LIN {X 0,Y 401.052,Z 702.53,A -85,B 0,C 180,E1 10289.297,E2 10289.297} C_VEL
LIN {X 0,Y 401.045,Z 702.53,A -85,B 0,C 180,E1 10294.373,E2 10294.373} C_VEL
LIN {X 0,Y 400.94,Z 702.53,A -85,B 0,C 180,E1 10301.171,E2 10301.171} C_VEL
LIN {X 0,Y 400.996,Z 702.775,A -85,B 0,C 180,E1 10303.002,E2 10303.002} C_VEL
LIN {X 0,Y 403.697,Z 708.428,A -85,B 0,C 180,E1 10303.533,E2 10303.533} C_VEL
LIN {X 0,Y 424.245,Z 745.989,A -85,B 0,C 180,E1 10307.047,E2 10307.047} C_VEL
LIN {X 0,Y 435.386,Z 772.98,A -85,B 0,C 180,E1 10309.087,E2 10309.087} C_VEL
LIN {X 0,Y 431.382,Z 812.336,A -85,B 0,C 180,E1 10310.627,E2 10310.627} C_VEL
LIN {X 0,Y 426.154,Z 850.577,A -85,B 0,C 180,E1 10312.988,E2 10312.988} C_VEL
LIN {X 0,Y 420.465,Z 885.103,A -85,B 0,C 180,E1 10316.006,E2 10316.006} C_VEL
LIN {X 0,Y 414.847,Z 916.19,A -85,B 0,C 180,E1 10319.673,E2 10319.673} C_VEL
LIN {X 0,Y 409.958,Z 944.249,A -85,B 0,C 180,E1 10324.079,E2 10324.079} C_VEL
LIN {X 0,Y 406.182,Z 967.928,A -85,B 0,C 180,E1 10329.048,E2 10329.048} C_VEL
LIN {X 0,Y 405.097,Z 975.872,A -85,B 0,C 180,E1 10331.112,E2 10331.112} C_VEL
LIN {X 0,Y 400.257,Z 983.264,A -85,B 0,C 180,E1 10333.268,E2 10333.268} C_VEL
LIN {X 0,Y 395.701,Z 989.61,A -85,B 0,C 180,E1 10335.54,E2 10335.54} C_VEL
LIN {X 0,Y 395,Z 999.376,A -85,B 0,C 180,E1 10340.101,E2 10340.101} C_VEL
LIN {X 0,Y 394.611,Z 1006.165,A -85,B 0,C 180,E1 10345.613,E2 10345.613} C_VEL
LIN {X 0,Y 394.714,Z 1007.908,A -85,B 0,C 180,E1 10350,E2 10350} C_VEL
LIN {X 0,Y 394.611,Z 1006.224,A -85,B 0,C 180,E1 10354.386,E2 10354.386} C_VEL
LIN {X 0,Y 394.945,Z 999.516,A -85,B 0,C 180,E1 10359.9,E2 10359.9} C_VEL
LIN {X 0,Y 395.941,Z 987.247,A -85,B 0,C 180,E1 10365.473,E2 10365.473} C_VEL
LIN {X 0,Y 398.331,Z 968.706,A -85,B 0,C 180,E1 10371.093,E2 10371.093} C_VEL
LIN {X 0,Y 402.279,Z 945.825,A -85,B 0,C 180,E1 10376.109,E2 10376.109} C_VEL
LIN {X 0,Y 407.443,Z 918.337,A -85,B 0,C 180,E1 10380.614,E2 10380.614} C_VEL
LIN {X 0,Y 413.535,Z 886.366,A -85,B 0,C 180,E1 10384.518,E2 10384.518} C_VEL
LIN {X 0,Y 419.816,Z 850.978,A -85,B 0,C 180,E1 10387.666,E2 10387.666} C_VEL
LIN {X 0,Y 425.063,Z 815.15,A -85,B 0,C 180,E1 10389.921,E2 10389.921} C_VEL
LIN {X 0,Y 429.128,Z 778.016,A -85,B 0,C 180,E1 10391.452,E2 10391.452} C_VEL
LIN {X 0,Y 428.274,Z 771.788,A -85,B 0,C 180,E1 10391.794,E2 10391.794} C_VEL
LIN {X 0,Y 411.741,Z 736.797,A -85,B 0,C 180,E1 10394.654,E2 10394.654} C_VEL
LIN {X 0,Y 393.146,Z 703.935,A -85,B 0,C 180,E1 10397.845,E2 10397.845} C_VEL
LIN {X 0,Y 392.991,Z 702.53,A -85,B 0,C 180,E1 10398.003,E2 10398.003} C_VEL
LIN {X 0,Y 393.035,Z 702.53,A -85,B 0,C 180,E1 10404.824,E2 10404.824} C_VEL
LIN {X 0,Y 393.229,Z 702.53,A -85,B 0,C 180,E1 10410.062,E2 10410.062} C_VEL
LIN {X 0,Y 393.395,Z 702.53,A -85,B 0,C 180,E1 10417.43,E2 10417.43} C_VEL
LIN {X 0,Y 393.756,Z 702.53,A -85,B 0,C 180,E1 10424.424,E2 10424.424} C_VEL
LIN {X 0,Y 394.01,Z 702.53,A -85,B 0,C 180,E1 10431.172,E2 10431.172} C_VEL
LIN {X 0,Y 394.34,Z 702.53,A -85,B 0,C 180,E1 10437.79,E2 10437.79} C_VEL
LIN {X 0,Y 394.238,Z 702.53,A -85,B 0,C 180,E1 10444.372,E2 10444.372} C_VEL
LIN {X 0,Y 393.912,Z 702.53,A -85,B 0,C 180,E1 10451.022,E2 10451.022} C_VEL
LIN {X 0,Y 393.605,Z 702.53,A -85,B 0,C 180,E1 10457.838,E2 10457.838} C_VEL
LIN {X 0,Y 393.332,Z 702.53,A -85,B 0,C 180,E1 10464.936,E2 10464.936} C_VEL
LIN {X 0,Y 393.129,Z 702.53,A -85,B 0,C 180,E1 10472.477,E2 10472.477} C_VEL
LIN {X 0,Y 393.096,Z 702.53,A -85,B 0,C 180,E1 10479.847,E2 10479.847} C_VEL
LIN {X 0,Y 392.99,Z 702.53,A -85,B 0,C 180,E1 10486.81,E2 10486.81} C_VEL
LIN {X 0,Y 393.02,Z 702.53,A -85,B 0,C 180,E1 10493.688,E2 10493.688} C_VEL
LIN {X 0,Y 393.251,Z 702.53,A -85,B 0,C 180,E1 10500.076,E2 10500.076} C_VEL
LIN {X 0,Y 393.474,Z 702.53,A -85,B 0,C 180,E1 10507.449,E2 10507.449} C_VEL
LIN {X 0,Y 393.781,Z 702.53,A -85,B 0,C 180,E1 10515.001,E2 10515.001} C_VEL
LIN {X 0,Y 393.859,Z 703.393,A -85,B 0,C 180,E1 10515.424,E2 10515.424} C_VEL
LIN {X 0,Y 412.86,Z 740.827,A -85,B 0,C 180,E1 10519.002,E2 10519.002} C_VEL
LIN {X 0,Y 422.422,Z 766.343,A -85,B 0,C 180,E1 10521.39,E2 10521.39} C_VEL
LIN {X 0,Y 417.672,Z 802.69,A -85,B 0,C 180,E1 10523.68,E2 10523.68} C_VEL
LIN {X 0,Y 412.384,Z 834.554,A -85,B 0,C 180,E1 10526.591,E2 10526.591} C_VEL
LIN {X 0,Y 406.978,Z 863.399,A -85,B 0,C 180,E1 10530.239,E2 10530.239} C_VEL
LIN {X 0,Y 401.875,Z 889.304,A -85,B 0,C 180,E1 10534.775,E2 10534.775} C_VEL
LIN {X 0,Y 398.263,Z 909.402,A -85,B 0,C 180,E1 10539.735,E2 10539.735} C_VEL
LIN {X 0,Y 396.131,Z 923.775,A -85,B 0,C 180,E1 10544.89,E2 10544.89} C_VEL
LIN {X 0,Y 395.152,Z 932.764,A -85,B 0,C 180,E1 10550.103,E2 10550.103} C_VEL
LIN {X 0,Y 394.324,Z 936.627,A -85,B 0,C 180,E1 10554.895,E2 10554.895} C_VEL
LIN {X 0,Y 394.397,Z 936.365,A -85,B 0,C 180,E1 10559.829,E2 10559.829} C_VEL
LIN {X 0,Y 395.362,Z 931.57,A -85,B 0,C 180,E1 10564.927,E2 10564.927} C_VEL
LIN {X 0,Y 396.711,Z 920.884,A -85,B 0,C 180,E1 10570.511,E2 10570.511} C_VEL
LIN {X 0,Y 399.154,Z 906.168,A -85,B 0,C 180,E1 10575.371,E2 10575.371} C_VEL
LIN {X 0,Y 403.025,Z 886.025,A -85,B 0,C 180,E1 10580.064,E2 10580.064} C_VEL
LIN {X 0,Y 408.334,Z 860.251,A -85,B 0,C 180,E1 10584.393,E2 10584.393} C_VEL
LIN {X 0,Y 414.18,Z 830.081,A -85,B 0,C 180,E1 10588.051,E2 10588.051} C_VEL
LIN {X 0,Y 419.598,Z 797.291,A -85,B 0,C 180,E1 10590.879,E2 10590.879} C_VEL
LIN {X 0,Y 423.349,Z 767.496,A -85,B 0,C 180,E1 10592.719,E2 10592.719} C_VEL
LIN {X 0,Y 410.879,Z 735.408,A -85,B 0,C 180,E1 10595.919,E2 10595.919} C_VEL
LIN {X 0,Y 394.941,Z 706.911,A -85,B 0,C 180,E1 10599.107,E2 10599.107} C_VEL
LIN {X 0,Y 393.602,Z 702.53,A -85,B 0,C 180,E1 10599.553,E2 10599.553} C_VEL
LIN {X 0,Y 393.925,Z 702.53,A -85,B 0,C 180,E1 10606.733,E2 10606.733} C_VEL
LIN {X 0,Y 394.164,Z 702.53,A -85,B 0,C 180,E1 10613.424,E2 10613.424} C_VEL
LIN {X 0,Y 394.433,Z 702.53,A -85,B 0,C 180,E1 10620.018,E2 10620.018} C_VEL
LIN {X 0,Y 394.167,Z 702.53,A -85,B 0,C 180,E1 10626.611,E2 10626.611} C_VEL
LIN {X 0,Y 393.791,Z 702.53,A -85,B 0,C 180,E1 10633.307,E2 10633.307} C_VEL
LIN {X 0,Y 393.496,Z 702.53,A -85,B 0,C 180,E1 10640.204,E2 10640.204} C_VEL
LIN {X 0,Y 393.162,Z 702.53,A -85,B 0,C 180,E1 10647.437,E2 10647.437} C_VEL
LIN {X 0,Y 393.102,Z 702.53,A -85,B 0,C 180,E1 10652.521,E2 10652.521} C_VEL
LIN {X 0,Y 393.103,Z 702.53,A -85,B 0,C 180,E1 10659.847,E2 10659.847} C_VEL
LIN {X 0,Y 393.027,Z 702.53,A -85,B 0,C 180,E1 10661.782,E2 10661.782} C_VEL
LIN {X 0,Y 395.507,Z 708.258,A -85,B 0,C 180,E1 10662.321,E2 10662.321} C_VEL
LIN {X 0,Y 413.841,Z 740.209,A -85,B 0,C 180,E1 10665.645,E2 10665.645} C_VEL
LIN {X 0,Y 428.982,Z 774.179,A -85,B 0,C 180,E1 10668.462,E2 10668.462} C_VEL
LIN {X 0,Y 424.791,Z 813.732,A -85,B 0,C 180,E1 10670.072,E2 10670.072} C_VEL
LIN {X 0,Y 419.489,Z 850.623,A -85,B 0,C 180,E1 10672.403,E2 10672.403} C_VEL
LIN {X 0,Y 413.587,Z 884.412,A -85,B 0,C 180,E1 10675.4,E2 10675.4} C_VEL
LIN {X 0,Y 407.742,Z 915.374,A -85,B 0,C 180,E1 10679.102,E2 10679.102} C_VEL
LIN {X 0,Y 402.477,Z 943.473,A -85,B 0,C 180,E1 10683.582,E2 10683.582} C_VEL
LIN {X 0,Y 398.489,Z 967.095,A -85,B 0,C 180,E1 10688.624,E2 10688.624} C_VEL
LIN {X 0,Y 396.091,Z 985.35,A -85,B 0,C 180,E1 10693.966,E2 10693.966} C_VEL
LIN {X 0,Y 395.701,Z 989.61,A -85,B 0,C 180,E1 10695.54,E2 10695.54} C_VEL
LIN {X 0,Y 394.194,Z 992.52,A -85,B 0,C 180,E1 10696.72,E2 10696.72} C_VEL
LIN {X 0,Y 387.214,Z 998.831,A -85,B 0,C 180,E1 10700.006,E2 10700.006} C_VEL
LIN {X 0,Y 387.072,Z 999.295,A -85,B 0,C 180,E1 10700.323,E2 10700.323} C_VEL
LIN {X 0,Y 386.742,Z 1005.449,A -85,B 0,C 180,E1 10705.524,E2 10705.524} C_VEL
LIN {X 0,Y 386.851,Z 1007.204,A -85,B 0,C 180,E1 10710,E2 10710} C_VEL
LIN {X 0,Y 386.743,Z 1005.522,A -85,B 0,C 180,E1 10714.475,E2 10714.475} C_VEL
LIN {X 0,Y 387.089,Z 998.806,A -85,B 0,C 180,E1 10720.103,E2 10720.103} C_VEL
LIN {X 0,Y 388.126,Z 986.517,A -85,B 0,C 180,E1 10725.792,E2 10725.792} C_VEL
LIN {X 0,Y 390.553,Z 968.854,A -85,B 0,C 180,E1 10731.294,E2 10731.294} C_VEL
LIN {X 0,Y 394.713,Z 946.035,A -85,B 0,C 180,E1 10736.443,E2 10736.443} C_VEL
LIN {X 0,Y 399.964,Z 919.435,A -85,B 0,C 180,E1 10740.934,E2 10740.934} C_VEL
LIN {X 0,Y 406.318,Z 887.704,A -85,B 0,C 180,E1 10744.929,E2 10744.929} C_VEL
LIN {X 0,Y 412.869,Z 852.832,A -85,B 0,C 180,E1 10748.128,E2 10748.128} C_VEL
LIN {X 0,Y 418.434,Z 816.703,A -85,B 0,C 180,E1 10750.477,E2 10750.477} C_VEL
LIN {X 0,Y 422.744,Z 779.639,A -85,B 0,C 180,E1 10752.058,E2 10752.058} C_VEL
LIN {X 0,Y 421.436,Z 773.287,A -85,B 0,C 180,E1 10752.464,E2 10752.464} C_VEL
LIN {X 0,Y 405.117,Z 738.587,A -85,B 0,C 180,E1 10755.43,E2 10755.43} C_VEL
LIN {X 0,Y 385.128,Z 703.353,A -85,B 0,C 180,E1 10759.006,E2 10759.006} C_VEL
LIN {X 0,Y 385.086,Z 702.53,A -85,B 0,C 180,E1 10759.18,E2 10759.18} C_VEL
LIN {X 0,Y 385.15,Z 702.53,A -85,B 0,C 180,E1 10766.722,E2 10766.722} C_VEL
LIN {X 0,Y 385.311,Z 702.53,A -85,B 0,C 180,E1 10771.955,E2 10771.955} C_VEL
LIN {X 0,Y 385.568,Z 702.53,A -85,B 0,C 180,E1 10779.362,E2 10779.362} C_VEL
LIN {X 0,Y 385.931,Z 702.53,A -85,B 0,C 180,E1 10786.416,E2 10786.416} C_VEL
LIN {X 0,Y 386.238,Z 702.53,A -85,B 0,C 180,E1 10793.252,E2 10793.252} C_VEL
LIN {X 0,Y 386.529,Z 702.53,A -85,B 0,C 180,E1 10799.982,E2 10799.982} C_VEL
LIN {X 0,Y 386.294,Z 702.53,A -85,B 0,C 180,E1 10806.71,E2 10806.71} C_VEL
LIN {X 0,Y 385.902,Z 702.53,A -85,B 0,C 180,E1 10813.548,E2 10813.548} C_VEL
LIN {X 0,Y 385.558,Z 702.53,A -85,B 0,C 180,E1 10820.601,E2 10820.601} C_VEL
LIN {X 0,Y 385.293,Z 702.53,A -85,B 0,C 180,E1 10828.006,E2 10828.006} C_VEL
LIN {X 0,Y 385.138,Z 702.53,A -85,B 0,C 180,E1 10835.963,E2 10835.963} C_VEL
LIN {X 0,Y 385.054,Z 702.53,A -85,B 0,C 180,E1 10841.875,E2 10841.875} C_VEL
LIN {X 0,Y 384.996,Z 702.53,A -85,B 0,C 180,E1 10848.216,E2 10848.216} C_VEL
LIN {X 0,Y 385.102,Z 702.53,A -85,B 0,C 180,E1 10855.323,E2 10855.323} C_VEL
LIN {X 0,Y 385.351,Z 702.53,A -85,B 0,C 180,E1 10861.971,E2 10861.971} C_VEL
LIN {X 0,Y 385.614,Z 702.53,A -85,B 0,C 180,E1 10869.379,E2 10869.379} C_VEL
LIN {X 0,Y 385.816,Z 702.53,A -85,B 0,C 180,E1 10874.301,E2 10874.301} C_VEL
LIN {X 0,Y 388.288,Z 708.228,A -85,B 0,C 180,E1 10874.797,E2 10874.797} C_VEL
LIN {X 0,Y 405.008,Z 740.357,A -85,B 0,C 180,E1 10878.064,E2 10878.064} C_VEL
LIN {X 0,Y 415.924,Z 768.941,A -85,B 0,C 180,E1 10880.868,E2 10880.868} C_VEL
LIN {X 0,Y 410.983,Z 804.002,A -85,B 0,C 180,E1 10883.128,E2 10883.128} C_VEL
LIN {X 0,Y 405.406,Z 836.162,A -85,B 0,C 180,E1 10886.132,E2 10886.132} C_VEL
LIN {X 0,Y 399.504,Z 865.889,A -85,B 0,C 180,E1 10890,E2 10890} C_VEL
LIN {X 0,Y 394.476,Z 890.181,A -85,B 0,C 180,E1 10894.388,E2 10894.388} C_VEL
LIN {X 0,Y 390.81,Z 909.432,A -85,B 0,C 180,E1 10899.202,E2 10899.202} C_VEL
LIN {X 0,Y 388.573,Z 922.95,A -85,B 0,C 180,E1 10903.991,E2 10903.991} C_VEL
LIN {X 0,Y 387.394,Z 932.609,A -85,B 0,C 180,E1 10909.336,E2 10909.336} C_VEL
LIN {X 0,Y 386.659,Z 936.306,A -85,B 0,C 180,E1 10912.972,E2 10912.972} C_VEL
LIN {X 0,Y 386.357,Z 937.678,A -85,B 0,C 180,E1 10917.95,E2 10917.95} C_VEL
LIN {X 0,Y 387.131,Z 934.693,A -85,B 0,C 180,E1 10923.074,E2 10923.074} C_VEL
LIN {X 0,Y 388.244,Z 926.715,A -85,B 0,C 180,E1 10928.454,E2 10928.454} C_VEL
LIN {X 0,Y 390.598,Z 912.563,A -85,B 0,C 180,E1 10934.06,E2 10934.06} C_VEL
LIN {X 0,Y 394.279,Z 894.078,A -85,B 0,C 180,E1 10938.972,E2 10938.972} C_VEL
LIN {X 0,Y 399.378,Z 870.198,A -85,B 0,C 180,E1 10943.524,E2 10943.524} C_VEL
LIN {X 0,Y 405.483,Z 841.302,A -85,B 0,C 180,E1 10947.501,E2 10947.501} C_VEL
LIN {X 0,Y 411.391,Z 809.409,A -85,B 0,C 180,E1 10950.634,E2 10950.634} C_VEL
LIN {X 0,Y 416.625,Z 774.543,A -85,B 0,C 180,E1 10953.01,E2 10953.01} C_VEL
LIN {X 0,Y 416.614,Z 769.06,A -85,B 0,C 180,E1 10953.395,E2 10953.395} C_VEL
LIN {X 0,Y 403.971,Z 736.735,A -85,B 0,C 180,E1 10956.786,E2 10956.786} C_VEL
LIN {X 0,Y 387.934,Z 707.99,A -85,B 0,C 180,E1 10960.187,E2 10960.187} C_VEL
LIN {X 0,Y 385.683,Z 702.53,A -85,B 0,C 180,E1 10960.896,E2 10960.896} C_VEL
LIN {X 0,Y 385.992,Z 702.53,A -85,B 0,C 180,E1 10967.789,E2 10967.789} C_VEL
LIN {X 0,Y 386.238,Z 702.53,A -85,B 0,C 180,E1 10973.289,E2 10973.289} C_VEL
LIN {X 0,Y 386.53,Z 702.53,A -85,B 0,C 180,E1 10980.018,E2 10980.018} C_VEL
LIN {X 0,Y 386.235,Z 702.53,A -85,B 0,C 180,E1 10986.748,E2 10986.748} C_VEL
LIN {X 0,Y 385.852,Z 702.53,A -85,B 0,C 180,E1 10993.586,E2 10993.586} C_VEL
LIN {X 0,Y 385.553,Z 702.53,A -85,B 0,C 180,E1 11000.639,E2 11000.639} C_VEL
LIN {X 0,Y 385.223,Z 702.53,A -85,B 0,C 180,E1 11008.052,E2 11008.052} C_VEL
LIN {X 0,Y 385.146,Z 702.53,A -85,B 0,C 180,E1 11016.007,E2 11016.007} C_VEL
LIN {X 0,Y 385.18,Z 702.898,A -85,B 0,C 180,E1 11020.512,E2 11020.512} C_VEL
LIN {X 0,Y 387.829,Z 708.463,A -85,B 0,C 180,E1 11021.108,E2 11021.108} C_VEL
LIN {X 0,Y 406.292,Z 740.05,A -85,B 0,C 180,E1 11024.654,E2 11024.654} C_VEL
LIN {X 0,Y 421.611,Z 774.151,A -85,B 0,C 180,E1 11027.65,E2 11027.65} C_VEL
LIN {X 0,Y 422.381,Z 779.875,A -85,B 0,C 180,E1 11027.975,E2 11027.975} C_VEL
LIN {X 0,Y 417.605,Z 820.164,A -85,B 0,C 180,E1 11029.765,E2 11029.765} C_VEL
LIN {X 0,Y 411.461,Z 858.485,A -85,B 0,C 180,E1 11032.41,E2 11032.41} C_VEL
LIN {X 0,Y 404.911,Z 893.328,A -85,B 0,C 180,E1 11035.82,E2 11035.82} C_VEL
LIN {X 0,Y 398.761,Z 924.07,A -85,B 0,C 180,E1 11039.906,E2 11039.906} C_VEL
LIN {X 0,Y 393.777,Z 950.025,A -85,B 0,C 180,E1 11044.502,E2 11044.502} C_VEL
LIN {X 0,Y 390.004,Z 972.744,A -85,B 0,C 180,E1 11049.916,E2 11049.916} C_VEL
LIN {X 0,Y 387.834,Z 989.469,A -85,B 0,C 180,E1 11055.496,E2 11055.496} C_VEL
LIN {X 0,Y 387.072,Z 999.295,A -85,B 0,C 180,E1 11060.323,E2 11060.323} C_VEL
LIN {X 0,Y 384.316,Z 1001.907,A -85,B 0,C 180,E1 11062.194,E2 11062.194} C_VEL
LIN {X 0,Y 378.936,Z 1004.429,A -85,B 0,C 180,E1 11065.042,E2 11065.042} C_VEL
LIN {X 0,Y 378.858,Z 1004.683,A -85,B 0,C 180,E1 11065.372,E2 11065.372} C_VEL
LIN {X 0,Y 379.004,Z 1006.502,A -85,B 0,C 180,E1 11070,E2 11070} C_VEL
LIN {X 0,Y 378.853,Z 1004.312,A -85,B 0,C 180,E1 11075.211,E2 11075.211} C_VEL
LIN {X 0,Y 379.22,Z 998.094,A -85,B 0,C 180,E1 11080.315,E2 11080.315} C_VEL
LIN {X 0,Y 380.331,Z 985.782,A -85,B 0,C 180,E1 11086.125,E2 11086.125} C_VEL
LIN {X 0,Y 382.881,Z 968.389,A -85,B 0,C 180,E1 11091.661,E2 11091.661} C_VEL
LIN {X 0,Y 387.43,Z 944.7,A -85,B 0,C 180,E1 11097.087,E2 11097.087} C_VEL
LIN {X 0,Y 393.311,Z 916.554,A -85,B 0,C 180,E1 11101.84,E2 11101.84} C_VEL
LIN {X 0,Y 399.792,Z 885.783,A -85,B 0,C 180,E1 11105.703,E2 11105.703} C_VEL
LIN {X 0,Y 406.534,Z 850.972,A -85,B 0,C 180,E1 11108.895,E2 11108.895} C_VEL
LIN {X 0,Y 412.45,Z 814.023,A -85,B 0,C 180,E1 11111.271,E2 11111.271} C_VEL
LIN {X 0,Y 416.104,Z 778.562,A -85,B 0,C 180,E1 11112.831,E2 11112.831} C_VEL
LIN {X 0,Y 400.377,Z 744.039,A -85,B 0,C 180,E1 11115.905,E2 11115.905} C_VEL
LIN {X 0,Y 379.039,Z 707.666,A -85,B 0,C 180,E1 11119.803,E2 11119.803} C_VEL
LIN {X 0,Y 377.121,Z 702.53,A -85,B 0,C 180,E1 11120.314,E2 11120.314} C_VEL
LIN {X 0,Y 377.215,Z 702.53,A -85,B 0,C 180,E1 11127.149,E2 11127.149} C_VEL
LIN {X 0,Y 377.396,Z 702.53,A -85,B 0,C 180,E1 11133.893,E2 11133.893} C_VEL
LIN {X 0,Y 377.729,Z 702.53,A -85,B 0,C 180,E1 11141.347,E2 11141.347} C_VEL
LIN {X 0,Y 378.103,Z 702.53,A -85,B 0,C 180,E1 11148.473,E2 11148.473} C_VEL
LIN {X 0,Y 378.469,Z 702.53,A -85,B 0,C 180,E1 11155.409,E2 11155.409} C_VEL
LIN {X 0,Y 378.657,Z 702.53,A -85,B 0,C 180,E1 11162.265,E2 11162.265} C_VEL
LIN {X 0,Y 378.162,Z 702.53,A -85,B 0,C 180,E1 11169.164,E2 11169.164} C_VEL
LIN {X 0,Y 377.779,Z 702.53,A -85,B 0,C 180,E1 11176.531,E2 11176.531} C_VEL
LIN {X 0,Y 377.492,Z 702.53,A -85,B 0,C 180,E1 11183.537,E2 11183.537} C_VEL
LIN {X 0,Y 377.307,Z 702.53,A -85,B 0,C 180,E1 11188.653,E2 11188.653} C_VEL
LIN {X 0,Y 377.186,Z 702.53,A -85,B 0,C 180,E1 11194.032,E2 11194.032} C_VEL
LIN {X 0,Y 377.092,Z 702.53,A -85,B 0,C 180,E1 11200.507,E2 11200.507} C_VEL
LIN {X 0,Y 377.001,Z 702.53,A -85,B 0,C 180,E1 11207.121,E2 11207.121} C_VEL
LIN {X 0,Y 377.151,Z 702.53,A -85,B 0,C 180,E1 11213.118,E2 11213.118} C_VEL
LIN {X 0,Y 377.258,Z 702.53,A -85,B 0,C 180,E1 11218.668,E2 11218.668} C_VEL
LIN {X 0,Y 377.48,Z 702.53,A -85,B 0,C 180,E1 11223.913,E2 11223.913} C_VEL
LIN {X 0,Y 377.655,Z 702.53,A -85,B 0,C 180,E1 11228.923,E2 11228.923} C_VEL
LIN {X 0,Y 377.773,Z 702.53,A -85,B 0,C 180,E1 11233.124,E2 11233.124} C_VEL
LIN {X 0,Y 380.209,Z 708.177,A -85,B 0,C 180,E1 11233.653,E2 11233.653} C_VEL
LIN {X 0,Y 397.132,Z 739.649,A -85,B 0,C 180,E1 11237.064,E2 11237.064} C_VEL
LIN {X 0,Y 409.133,Z 770.794,A -85,B 0,C 180,E1 11240.249,E2 11240.249} C_VEL
LIN {X 0,Y 404.201,Z 806.198,A -85,B 0,C 180,E1 11242.632,E2 11242.632} C_VEL
LIN {X 0,Y 398.183,Z 838.981,A -85,B 0,C 180,E1 11245.789,E2 11245.789} C_VEL
LIN {X 0,Y 392.138,Z 867.822,A -85,B 0,C 180,E1 11249.685,E2 11249.685} C_VEL
LIN {X 0,Y 386.888,Z 891.998,A -85,B 0,C 180,E1 11254.194,E2 11254.194} C_VEL
LIN {X 0,Y 383.102,Z 910.836,A -85,B 0,C 180,E1 11259.066,E2 11259.066} C_VEL
LIN {X 0,Y 380.653,Z 924.901,A -85,B 0,C 180,E1 11264.288,E2 11264.288} C_VEL
LIN {X 0,Y 379.481,Z 934.068,A -85,B 0,C 180,E1 11269.756,E2 11269.756} C_VEL
LIN {X 0,Y 378.675,Z 937.5,A -85,B 0,C 180,E1 11273.65,E2 11273.65} C_VEL
LIN {X 0,Y 378.509,Z 938.284,A -85,B 0,C 180,E1 11278.77,E2 11278.77} C_VEL
LIN {X 0,Y 379.648,Z 933.538,A -85,B 0,C 180,E1 11284.869,E2 11284.869} C_VEL
LIN {X 0,Y 380.883,Z 924.814,A -85,B 0,C 180,E1 11289.991,E2 11289.991} C_VEL
LIN {X 0,Y 383.757,Z 909.485,A -85,B 0,C 180,E1 11295.609,E2 11295.609} C_VEL
LIN {X 0,Y 388.144,Z 889.289,A -85,B 0,C 180,E1 11300.662,E2 11300.662} C_VEL
LIN {X 0,Y 393.75,Z 864.896,A -85,B 0,C 180,E1 11305.023,E2 11305.023} C_VEL
LIN {X 0,Y 399.996,Z 835.936,A -85,B 0,C 180,E1 11308.798,E2 11308.798} C_VEL
LIN {X 0,Y 406.42,Z 802.058,A -85,B 0,C 180,E1 11311.934,E2 11311.934} C_VEL
LIN {X 0,Y 410.569,Z 772.881,A -85,B 0,C 180,E1 11313.854,E2 11313.854} C_VEL
LIN {X 0,Y 398.541,Z 741.008,A -85,B 0,C 180,E1 11317.337,E2 11317.337} C_VEL
LIN {X 0,Y 383.43,Z 713.411,A -85,B 0,C 180,E1 11320.772,E2 11320.772} C_VEL
LIN {X 0,Y 377.87,Z 703.299,A -85,B 0,C 180,E1 11322.07,E2 11322.07} C_VEL
LIN {X 0,Y 378.151,Z 702.53,A -85,B 0,C 180,E1 11328.512,E2 11328.512} C_VEL
LIN {X 0,Y 378.433,Z 702.53,A -85,B 0,C 180,E1 11335.485,E2 11335.485} C_VEL
LIN {X 0,Y 378.66,Z 702.53,A -85,B 0,C 180,E1 11342.302,E2 11342.302} C_VEL
LIN {X 0,Y 378.107,Z 702.53,A -85,B 0,C 180,E1 11349.202,E2 11349.202} C_VEL
LIN {X 0,Y 377.748,Z 702.53,A -85,B 0,C 180,E1 11356.513,E2 11356.513} C_VEL
LIN {X 0,Y 377.496,Z 702.53,A -85,B 0,C 180,E1 11363.576,E2 11363.576} C_VEL
LIN {X 0,Y 377.262,Z 702.53,A -85,B 0,C 180,E1 11368.698,E2 11368.698} C_VEL
LIN {X 0,Y 377.169,Z 702.53,A -85,B 0,C 180,E1 11374.078,E2 11374.078} C_VEL
LIN {X 0,Y 377.286,Z 702.53,A -85,B 0,C 180,E1 11379.06,E2 11379.06} C_VEL
LIN {X 0,Y 379.809,Z 708.304,A -85,B 0,C 180,E1 11379.729,E2 11379.729} C_VEL
LIN {X 0,Y 397.649,Z 737.953,A -85,B 0,C 180,E1 11383.395,E2 11383.395} C_VEL
LIN {X 0,Y 413.023,Z 770.6,A -85,B 0,C 180,E1 11386.493,E2 11386.493} C_VEL
LIN {X 0,Y 416.247,Z 780.555,A -85,B 0,C 180,E1 11387.307,E2 11387.307} C_VEL
LIN {X 0,Y 411.1,Z 821.27,A -85,B 0,C 180,E1 11389.168,E2 11389.168} C_VEL
LIN {X 0,Y 404.613,Z 859.536,A -85,B 0,C 180,E1 11391.88,E2 11391.88} C_VEL
LIN {X 0,Y 397.83,Z 893.812,A -85,B 0,C 180,E1 11395.321,E2 11395.321} C_VEL
LIN {X 0,Y 391.626,Z 923.179,A -85,B 0,C 180,E1 11399.299,E2 11399.299} C_VEL
LIN {X 0,Y 386.205,Z 949.802,A -85,B 0,C 180,E1 11404.103,E2 11404.103} C_VEL
LIN {X 0,Y 382.283,Z 971.93,A -85,B 0,C 180,E1 11409.492,E2 11409.492} C_VEL
LIN {X 0,Y 380.048,Z 988.341,A -85,B 0,C 180,E1 11415.043,E2 11415.043} C_VEL
LIN {X 0,Y 379.113,Z 999.65,A -85,B 0,C 180,E1 11420.838,E2 11420.838} C_VEL
LIN {X 0,Y 378.858,Z 1004.683,A -85,B 0,C 180,E1 11425.372,E2 11425.372} C_VEL
LIN {X 0,Y 376.468,Z 1005.716,A -85,B 0,C 180,E1 11427.316,E2 11427.316} C_VEL
LIN {X 0,Y 371.069,Z 1005.689,A -85,B 0,C 180,E1 11430.597,E2 11430.597} C_VEL
LIN {X 0,Y 370.976,Z 1003.608,A -85,B 0,C 180,E1 11435.322,E2 11435.322} C_VEL
LIN {X 0,Y 371.343,Z 997.378,A -85,B 0,C 180,E1 11440.536,E2 11440.536} C_VEL
LIN {X 0,Y 372.553,Z 985.045,A -85,B 0,C 180,E1 11446.471,E2 11446.471} C_VEL
LIN {X 0,Y 375.517,Z 966.464,A -85,B 0,C 180,E1 11452.427,E2 11452.427} C_VEL
LIN {X 0,Y 380.219,Z 943.143,A -85,B 0,C 180,E1 11457.796,E2 11457.796} C_VEL
LIN {X 0,Y 386.343,Z 915.654,A -85,B 0,C 180,E1 11462.484,E2 11462.484} C_VEL
LIN {X 0,Y 393.17,Z 884.67,A -85,B 0,C 180,E1 11466.408,E2 11466.408} C_VEL
LIN {X 0,Y 400.185,Z 849.741,A -85,B 0,C 180,E1 11469.632,E2 11469.632} C_VEL
LIN {X 0,Y 406.418,Z 812.024,A -85,B 0,C 180,E1 11472.055,E2 11472.055} C_VEL
LIN {X 0,Y 409.801,Z 781.319,A -85,B 0,C 180,E1 11473.428,E2 11473.428} C_VEL
LIN {X 0,Y 394.34,Z 747.033,A -85,B 0,C 180,E1 11476.606,E2 11476.606} C_VEL
LIN {X 0,Y 371.535,Z 708.11,A -85,B 0,C 180,E1 11480.967,E2 11480.967} C_VEL
LIN {X 0,Y 369.264,Z 702.53,A -85,B 0,C 180,E1 11481.607,E2 11481.607} C_VEL
LIN {X 0,Y 369.337,Z 702.53,A -85,B 0,C 180,E1 11489.093,E2 11489.093} C_VEL
LIN {X 0,Y 369.521,Z 702.53,A -85,B 0,C 180,E1 11495.883,E2 11495.883} C_VEL
LIN {X 0,Y 369.912,Z 702.53,A -85,B 0,C 180,E1 11503.392,E2 11503.392} C_VEL
LIN {X 0,Y 370.221,Z 702.53,A -85,B 0,C 180,E1 11510.6,E2 11510.6} C_VEL
LIN {X 0,Y 370.642,Z 702.53,A -85,B 0,C 180,E1 11517.648,E2 11517.648} C_VEL
LIN {X 0,Y 370.754,Z 702.53,A -85,B 0,C 180,E1 11522.313,E2 11522.313} C_VEL
LIN {X 0,Y 370.23,Z 702.53,A -85,B 0,C 180,E1 11529.362,E2 11529.362} C_VEL
LIN {X 0,Y 369.88,Z 702.53,A -85,B 0,C 180,E1 11536.57,E2 11536.57} C_VEL
LIN {X 0,Y 369.506,Z 702.53,A -85,B 0,C 180,E1 11544.077,E2 11544.077} C_VEL
LIN {X 0,Y 369.276,Z 702.53,A -85,B 0,C 180,E1 11552.058,E2 11552.058} C_VEL
LIN {X 0,Y 369.151,Z 702.53,A -85,B 0,C 180,E1 11559.042,E2 11559.042} C_VEL
LIN {X 0,Y 369.103,Z 702.53,A -85,B 0,C 180,E1 11565.972,E2 11565.972} C_VEL
LIN {X 0,Y 369.14,Z 702.53,A -85,B 0,C 180,E1 11572.18,E2 11572.18} C_VEL
LIN {X 0,Y 369.349,Z 702.53,A -85,B 0,C 180,E1 11579.032,E2 11579.032} C_VEL
LIN {X 0,Y 369.61,Z 702.53,A -85,B 0,C 180,E1 11585.904,E2 11585.904} C_VEL
LIN {X 0,Y 369.822,Z 702.53,A -85,B 0,C 180,E1 11591.921,E2 11591.921} C_VEL
LIN {X 0,Y 372.289,Z 708.244,A -85,B 0,C 180,E1 11592.473,E2 11592.473} C_VEL
LIN {X 0,Y 389.277,Z 739.126,A -85,B 0,C 180,E1 11596.024,E2 11596.024} C_VEL
LIN {X 0,Y 401.577,Z 770.146,A -85,B 0,C 180,E1 11599.338,E2 11599.338} C_VEL
LIN {X 0,Y 402.569,Z 775.904,A -85,B 0,C 180,E1 11599.864,E2 11599.864} C_VEL
LIN {X 0,Y 396.964,Z 811.27,A -85,B 0,C 180,E1 11602.354,E2 11602.354} C_VEL
LIN {X 0,Y 390.438,Z 843.936,A -85,B 0,C 180,E1 11605.706,E2 11605.706} C_VEL
LIN {X 0,Y 384.153,Z 872.532,A -85,B 0,C 180,E1 11609.821,E2 11609.821} C_VEL
LIN {X 0,Y 378.711,Z 896.377,A -85,B 0,C 180,E1 11614.571,E2 11614.571} C_VEL
LIN {X 0,Y 374.695,Z 915.508,A -85,B 0,C 180,E1 11620.009,E2 11620.009} C_VEL
LIN {X 0,Y 372.52,Z 928.057,A -85,B 0,C 180,E1 11625.267,E2 11625.267} C_VEL
LIN {X 0,Y 371.573,Z 935.124,A -85,B 0,C 180,E1 11629.937,E2 11629.937} C_VEL
LIN {X 0,Y 370.763,Z 938.399,A -85,B 0,C 180,E1 11634.017,E2 11634.017} C_VEL
LIN {X 0,Y 370.681,Z 938.831,A -85,B 0,C 180,E1 11639.243,E2 11639.243} C_VEL
LIN {X 0,Y 371.756,Z 934.783,A -85,B 0,C 180,E1 11644.631,E2 11644.631} C_VEL
LIN {X 0,Y 373.185,Z 925.469,A -85,B 0,C 180,E1 11650.315,E2 11650.315} C_VEL
LIN {X 0,Y 376.253,Z 910.253,A -85,B 0,C 180,E1 11656.007,E2 11656.007} C_VEL
LIN {X 0,Y 381.161,Z 889.229,A -85,B 0,C 180,E1 11661.325,E2 11661.325} C_VEL
LIN {X 0,Y 386.936,Z 865.311,A -85,B 0,C 180,E1 11665.652,E2 11665.652} C_VEL
LIN {X 0,Y 393.585,Z 836.027,A -85,B 0,C 180,E1 11669.505,E2 11669.505} C_VEL
LIN {X 0,Y 400.314,Z 801.872,A -85,B 0,C 180,E1 11672.683,E2 11672.683} C_VEL
LIN {X 0,Y 404.144,Z 775.298,A -85,B 0,C 180,E1 11674.478,E2 11674.478} C_VEL
LIN {X 0,Y 392.631,Z 744.135,A -85,B 0,C 180,E1 11678.043,E2 11678.043} C_VEL
LIN {X 0,Y 376.909,Z 714.923,A -85,B 0,C 180,E1 11681.872,E2 11681.872} C_VEL
LIN {X 0,Y 370.151,Z 704.088,A -85,B 0,C 180,E1 11683.518,E2 11683.518} C_VEL
LIN {X 0,Y 370.054,Z 702.53,A -85,B 0,C 180,E1 11683.742,E2 11683.742} C_VEL
LIN {X 0,Y 370.256,Z 702.53,A -85,B 0,C 180,E1 11690.639,E2 11690.639} C_VEL
LIN {X 0,Y 370.584,Z 702.53,A -85,B 0,C 180,E1 11697.686,E2 11697.686} C_VEL
LIN {X 0,Y 370.757,Z 702.53,A -85,B 0,C 180,E1 11702.351,E2 11702.351} C_VEL
LIN {X 0,Y 370.174,Z 702.53,A -85,B 0,C 180,E1 11709.401,E2 11709.401} C_VEL
LIN {X 0,Y 369.844,Z 702.53,A -85,B 0,C 180,E1 11716.611,E2 11716.611} C_VEL
LIN {X 0,Y 369.502,Z 702.53,A -85,B 0,C 180,E1 11724.119,E2 11724.119} C_VEL
LIN {X 0,Y 369.235,Z 702.53,A -85,B 0,C 180,E1 11732.107,E2 11732.107} C_VEL
LIN {X 0,Y 369.312,Z 702.53,A -85,B 0,C 180,E1 11737.548,E2 11737.548} C_VEL
LIN {X 0,Y 371.458,Z 707.855,A -85,B 0,C 180,E1 11738.15,E2 11738.15} C_VEL
LIN {X 0,Y 386.545,Z 731.353,A -85,B 0,C 180,E1 11741.519,E2 11741.519} C_VEL
LIN {X 0,Y 403.453,Z 764.901,A -85,B 0,C 180,E1 11745.054,E2 11745.054} C_VEL
LIN {X 0,Y 409.937,Z 783.316,A -85,B 0,C 180,E1 11746.694,E2 11746.694} C_VEL
LIN {X 0,Y 404.617,Z 822.595,A -85,B 0,C 180,E1 11748.565,E2 11748.565} C_VEL
LIN {X 0,Y 398.086,Z 859.155,A -85,B 0,C 180,E1 11751.205,E2 11751.205} C_VEL
LIN {X 0,Y 391.063,Z 892.891,A -85,B 0,C 180,E1 11754.632,E2 11754.632} C_VEL
LIN {X 0,Y 384.57,Z 922.32,A -85,B 0,C 180,E1 11758.673,E2 11758.673} C_VEL
LIN {X 0,Y 378.686,Z 949.58,A -85,B 0,C 180,E1 11763.691,E2 11763.691} C_VEL
LIN {X 0,Y 374.573,Z 971.125,A -85,B 0,C 180,E1 11769.05,E2 11769.05} C_VEL
LIN {X 0,Y 372.22,Z 987.57,A -85,B 0,C 180,E1 11774.721,E2 11774.721} C_VEL
LIN {X 0,Y 371.407,Z 997.144,A -85,B 0,C 180,E1 11779.465,E2 11779.465} C_VEL
LIN {X 0,Y 370.992,Z 1004.028,A -85,B 0,C 180,E1 11785.361,E2 11785.361} C_VEL
LIN {X 0,Y 371.069,Z 1005.689,A -85,B 0,C 180,E1 11790.597,E2 11790.597} C_VEL
LIN {X 0,Y 368.441,Z 1005.044,A -85,B 0,C 180,E1 11792.589,E2 11792.589} C_VEL
LIN {X 0,Y 363.191,Z 1002.807,A -85,B 0,C 180,E1 11795.581,E2 11795.581} C_VEL
LIN {X 0,Y 363.118,Z 1002.533,A -85,B 0,C 180,E1 11795.927,E2 11795.927} C_VEL
LIN {X 0,Y 363.671,Z 994.641,A -85,B 0,C 180,E1 11801.974,E2 11801.974} C_VEL
LIN {X 0,Y 365.363,Z 980.737,A -85,B 0,C 180,E1 11808.185,E2 11808.185} C_VEL
LIN {X 0,Y 369.163,Z 959.923,A -85,B 0,C 180,E1 11814.434,E2 11814.434} C_VEL
LIN {X 0,Y 374.423,Z 935.916,A -85,B 0,C 180,E1 11819.631,E2 11819.631} C_VEL
LIN {X 0,Y 381.34,Z 906.505,A -85,B 0,C 180,E1 11824.325,E2 11824.325} C_VEL
LIN {X 0,Y 388.788,Z 873.679,A -85,B 0,C 180,E1 11828.166,E2 11828.166} C_VEL
LIN {X 0,Y 395.649,Z 839.123,A -85,B 0,C 180,E1 11831.086,E2 11831.086} C_VEL
LIN {X 0,Y 401.483,Z 802.504,A -85,B 0,C 180,E1 11833.222,E2 11833.222} C_VEL
LIN {X 0,Y 403.248,Z 783.359,A -85,B 0,C 180,E1 11834.097,E2 11834.097} C_VEL
LIN {X 0,Y 387.829,Z 748.995,A -85,B 0,C 180,E1 11837.433,E2 11837.433} C_VEL
LIN {X 0,Y 363.879,Z 708.339,A -85,B 0,C 180,E1 11842.222,E2 11842.222} C_VEL
LIN {X 0,Y 361.304,Z 703.395,A -85,B 0,C 180,E1 11842.81,E2 11842.81} C_VEL
LIN {X 0,Y 361.233,Z 702.53,A -85,B 0,C 180,E1 11843.402,E2 11843.402} C_VEL
LIN {X 0,Y 361.416,Z 702.53,A -85,B 0,C 180,E1 11849.917,E2 11849.917} C_VEL
LIN {X 0,Y 361.677,Z 702.53,A -85,B 0,C 180,E1 11857.929,E2 11857.929} C_VEL
LIN {X 0,Y 362.085,Z 702.53,A -85,B 0,C 180,E1 11865.503,E2 11865.503} C_VEL
LIN {X 0,Y 362.474,Z 702.53,A -85,B 0,C 180,E1 11872.808,E2 11872.808} C_VEL
LIN {X 0,Y 362.848,Z 702.53,A -85,B 0,C 180,E1 11879.981,E2 11879.981} C_VEL
LIN {X 0,Y 362.525,Z 702.53,A -85,B 0,C 180,E1 11887.153,E2 11887.153} C_VEL
LIN {X 0,Y 362.053,Z 702.53,A -85,B 0,C 180,E1 11894.459,E2 11894.459} C_VEL
LIN {X 0,Y 361.662,Z 702.53,A -85,B 0,C 180,E1 11902.03,E2 11902.03} C_VEL
LIN {X 0,Y 361.357,Z 702.53,A -85,B 0,C 180,E1 11910.044,E2 11910.044} C_VEL
LIN {X 0,Y 361.239,Z 702.53,A -85,B 0,C 180,E1 11917.468,E2 11917.468} C_VEL
LIN {X 0,Y 361.181,Z 702.53,A -85,B 0,C 180,E1 11924.744,E2 11924.744} C_VEL
LIN {X 0,Y 361.193,Z 702.53,A -85,B 0,C 180,E1 11931.195,E2 11931.195} C_VEL
LIN {X 0,Y 361.307,Z 702.53,A -85,B 0,C 180,E1 11937.115,E2 11937.115} C_VEL
LIN {X 0,Y 361.503,Z 702.53,A -85,B 0,C 180,E1 11942.667,E2 11942.667} C_VEL
LIN {X 0,Y 361.727,Z 702.53,A -85,B 0,C 180,E1 11947.948,E2 11947.948} C_VEL
LIN {X 0,Y 361.859,Z 702.759,A -85,B 0,C 180,E1 11950.642,E2 11950.642} C_VEL
LIN {X 0,Y 364.38,Z 708.242,A -85,B 0,C 180,E1 11951.221,E2 11951.221} C_VEL
LIN {X 0,Y 381.847,Z 739.41,A -85,B 0,C 180,E1 11955.025,E2 11955.025} C_VEL
LIN {X 0,Y 394.07,Z 769.915,A -85,B 0,C 180,E1 11958.419,E2 11958.419} C_VEL
LIN {X 0,Y 396.07,Z 778.227,A -85,B 0,C 180,E1 11959.273,E2 11959.273} C_VEL
LIN {X 0,Y 390.134,Z 813.452,A -85,B 0,C 180,E1 11961.835,E2 11961.835} C_VEL
LIN {X 0,Y 383.467,Z 845.449,A -85,B 0,C 180,E1 11965.203,E2 11965.203} C_VEL
LIN {X 0,Y 376.84,Z 874.196,A -85,B 0,C 180,E1 11969.446,E2 11969.446} C_VEL
LIN {X 0,Y 371.064,Z 898.092,A -85,B 0,C 180,E1 11974.373,E2 11974.373} C_VEL
LIN {X 0,Y 367.112,Z 916.065,A -85,B 0,C 180,E1 11979.612,E2 11979.612} C_VEL
LIN {X 0,Y 364.758,Z 928.677,A -85,B 0,C 180,E1 11984.985,E2 11984.985} C_VEL
LIN {X 0,Y 363.645,Z 936.349,A -85,B 0,C 180,E1 11990.322,E2 11990.322} C_VEL
LIN {X 0,Y 362.813,Z 939.38,A -85,B 0,C 180,E1 11994.578,E2 11994.578} C_VEL
LIN {X 0,Y 362.894,Z 939.299,A -85,B 0,C 180,E1 11999.934,E2 11999.934} C_VEL
LIN {X 0,Y 364.035,Z 934.701,A -85,B 0,C 180,E1 12005.475,E2 12005.475} C_VEL
LIN {X 0,Y 365.784,Z 924.761,A -85,B 0,C 180,E1 12011.306,E2 12011.306} C_VEL
LIN {X 0,Y 369.155,Z 909.368,A -85,B 0,C 180,E1 12016.937,E2 12016.937} C_VEL
LIN {X 0,Y 374.157,Z 889.211,A -85,B 0,C 180,E1 12022.017,E2 12022.017} C_VEL
LIN {X 0,Y 380.344,Z 864.95,A -85,B 0,C 180,E1 12026.427,E2 12026.427} C_VEL
LIN {X 0,Y 387.226,Z 836.19,A -85,B 0,C 180,E1 12030.232,E2 12030.232} C_VEL
LIN {X 0,Y 394.011,Z 803.266,A -85,B 0,C 180,E1 12033.338,E2 12033.338} C_VEL
LIN {X 0,Y 397.94,Z 778.535,A -85,B 0,C 180,E1 12035.043,E2 12035.043} C_VEL
LIN {X 0,Y 387.131,Z 748.228,A -85,B 0,C 180,E1 12038.666,E2 12038.666} C_VEL
LIN {X 0,Y 372.642,Z 720.57,A -85,B 0,C 180,E1 12042.457,E2 12042.457} C_VEL
LIN {X 0,Y 364.408,Z 708.059,A -85,B 0,C 180,E1 12044.563,E2 12044.563} C_VEL
LIN {X 0,Y 362.164,Z 702.53,A -85,B 0,C 180,E1 12045.392,E2 12045.392} C_VEL
LIN {X 0,Y 362.475,Z 702.53,A -85,B 0,C 180,E1 12052.846,E2 12052.846} C_VEL
LIN {X 0,Y 362.848,Z 702.53,A -85,B 0,C 180,E1 12060.019,E2 12060.019} C_VEL
LIN {X 0,Y 362.464,Z 702.53,A -85,B 0,C 180,E1 12067.192,E2 12067.192} C_VEL
LIN {X 0,Y 362.015,Z 702.53,A -85,B 0,C 180,E1 12074.5,E2 12074.5} C_VEL
LIN {X 0,Y 361.664,Z 702.53,A -85,B 0,C 180,E1 12082.072,E2 12082.072} C_VEL
LIN {X 0,Y 361.318,Z 702.53,A -85,B 0,C 180,E1 12090.092,E2 12090.092} C_VEL
LIN {X 0,Y 361.312,Z 703.018,A -85,B 0,C 180,E1 12095.859,E2 12095.859} C_VEL
LIN {X 0,Y 363.911,Z 708.331,A -85,B 0,C 180,E1 12096.613,E2 12096.613} C_VEL
LIN {X 0,Y 373.665,Z 722.805,A -85,B 0,C 180,E1 12099.032,E2 12099.032} C_VEL
LIN {X 0,Y 390.199,Z 751.789,A -85,B 0,C 180,E1 12102.688,E2 12102.688} C_VEL
LIN {X 0,Y 403.695,Z 784.375,A -85,B 0,C 180,E1 12105.983,E2 12105.983} C_VEL
LIN {X 0,Y 398.424,Z 822.492,A -85,B 0,C 180,E1 12107.851,E2 12107.851} C_VEL
LIN {X 0,Y 391.54,Z 859.262,A -85,B 0,C 180,E1 12110.55,E2 12110.55} C_VEL
LIN {X 0,Y 384.1,Z 893.197,A -85,B 0,C 180,E1 12114.066,E2 12114.066} C_VEL
LIN {X 0,Y 377.026,Z 923.542,A -85,B 0,C 180,E1 12118.359,E2 12118.359} C_VEL
LIN {X 0,Y 370.915,Z 950.602,A -85,B 0,C 180,E1 12123.529,E2 12123.529} C_VEL
LIN {X 0,Y 366.495,Z 973.415,A -85,B 0,C 180,E1 12129.513,E2 12129.513} C_VEL
LIN {X 0,Y 364.098,Z 989.602,A -85,B 0,C 180,E1 12135.601,E2 12135.601} C_VEL
LIN {X 0,Y 363.276,Z 999.844,A -85,B 0,C 180,E1 12141.64,E2 12141.64} C_VEL
LIN {X 0,Y 363.159,Z 1004.61,A -85,B 0,C 180,E1 12147.618,E2 12147.618} C_VEL
LIN {X 0,Y 363.183,Z 1004.667,A -85,B 0,C 180,E1 12152.381,E2 12152.381} C_VEL
LIN {X 0,Y 363.118,Z 1002.533,A -85,B 0,C 180,E1 12155.927,E2 12155.927} C_VEL
LIN {X 0,Y 360.727,Z 1000.469,A -85,B 0,C 180,E1 12157.943,E2 12157.943} C_VEL
LIN {X 0,Y 355.727,Z 996.051,A -85,B 0,C 180,E1 12160.945,E2 12160.945} C_VEL
LIN {X 0,Y 355.686,Z 995.484,A -85,B 0,C 180,E1 12161.289,E2 12161.289} C_VEL
LIN {X 0,Y 357.05,Z 983.555,A -85,B 0,C 180,E1 12167.208,E2 12167.208} C_VEL
LIN {X 0,Y 360.304,Z 965.293,A -85,B 0,C 180,E1 12173.31,E2 12173.31} C_VEL
LIN {X 0,Y 365.315,Z 942.947,A -85,B 0,C 180,E1 12178.698,E2 12178.698} C_VEL
LIN {X 0,Y 371.916,Z 916.119,A -85,B 0,C 180,E1 12183.493,E2 12183.493} C_VEL
LIN {X 0,Y 379.432,Z 885.193,A -85,B 0,C 180,E1 12187.584,E2 12187.584} C_VEL
LIN {X 0,Y 386.84,Z 851.566,A -85,B 0,C 180,E1 12190.822,E2 12190.822} C_VEL
LIN {X 0,Y 393.364,Z 815.906,A -85,B 0,C 180,E1 12193.246,E2 12193.246} C_VEL
LIN {X 0,Y 396.915,Z 786.124,A -85,B 0,C 180,E1 12194.714,E2 12194.714} C_VEL
LIN {X 0,Y 381.864,Z 752.088,A -85,B 0,C 180,E1 12198.181,E2 12198.181} C_VEL
LIN {X 0,Y 359.563,Z 714.053,A -85,B 0,C 180,E1 12202.801,E2 12202.801} C_VEL
LIN {X 0,Y 353.402,Z 703.512,A -85,B 0,C 180,E1 12204.222,E2 12204.222} C_VEL
LIN {X 0,Y 353.288,Z 702.53,A -85,B 0,C 180,E1 12204.468,E2 12204.468} C_VEL
LIN {X 0,Y 353.502,Z 702.53,A -85,B 0,C 180,E1 12211.979,E2 12211.979} C_VEL
LIN {X 0,Y 353.833,Z 702.53,A -85,B 0,C 180,E1 12220.035,E2 12220.035} C_VEL
LIN {X 0,Y 354.293,Z 702.53,A -85,B 0,C 180,E1 12227.687,E2 12227.687} C_VEL
LIN {X 0,Y 354.714,Z 702.53,A -85,B 0,C 180,E1 12235.101,E2 12235.101} C_VEL
LIN {X 0,Y 354.94,Z 702.53,A -85,B 0,C 180,E1 12242.417,E2 12242.417} C_VEL
LIN {X 0,Y 354.365,Z 702.53,A -85,B 0,C 180,E1 12249.785,E2 12249.785} C_VEL
LIN {X 0,Y 353.964,Z 702.53,A -85,B 0,C 180,E1 12257.338,E2 12257.338} C_VEL
LIN {X 0,Y 353.572,Z 702.53,A -85,B 0,C 180,E1 12265.236,E2 12265.236} C_VEL
LIN {X 0,Y 353.328,Z 702.53,A -85,B 0,C 180,E1 12271.332,E2 12271.332} C_VEL
LIN {X 0,Y 353.302,Z 702.53,A -85,B 0,C 180,E1 12276.69,E2 12276.69} C_VEL
LIN {X 0,Y 353.181,Z 702.53,A -85,B 0,C 180,E1 12283.419,E2 12283.419} C_VEL
LIN {X 0,Y 353.219,Z 702.53,A -85,B 0,C 180,E1 12290.217,E2 12290.217} C_VEL
LIN {X 0,Y 353.35,Z 702.53,A -85,B 0,C 180,E1 12296.277,E2 12296.277} C_VEL
LIN {X 0,Y 353.569,Z 702.53,A -85,B 0,C 180,E1 12303.601,E2 12303.601} C_VEL
LIN {X 0,Y 353.808,Z 702.53,A -85,B 0,C 180,E1 12309.201,E2 12309.201} C_VEL
LIN {X 0,Y 356.282,Z 708.196,A -85,B 0,C 180,E1 12309.856,E2 12309.856} C_VEL
LIN {X 0,Y 373.535,Z 738.088,A -85,B 0,C 180,E1 12313.763,E2 12313.763} C_VEL
LIN {X 0,Y 386.39,Z 768.786,A -85,B 0,C 180,E1 12317.373,E2 12317.373} C_VEL
LIN {X 0,Y 389.615,Z 780.679,A -85,B 0,C 180,E1 12318.674,E2 12318.674} C_VEL
LIN {X 0,Y 383.301,Z 815.938,A -85,B 0,C 180,E1 12321.332,E2 12321.332} C_VEL
LIN {X 0,Y 376.527,Z 846.933,A -85,B 0,C 180,E1 12324.683,E2 12324.683} C_VEL
LIN {X 0,Y 369.843,Z 874.76,A -85,B 0,C 180,E1 12328.871,E2 12328.871} C_VEL
LIN {X 0,Y 363.754,Z 898.53,A -85,B 0,C 180,E1 12333.841,E2 12333.841} C_VEL
LIN {X 0,Y 359.661,Z 916.153,A -85,B 0,C 180,E1 12339.032,E2 12339.032} C_VEL
LIN {X 0,Y 357.014,Z 929.293,A -85,B 0,C 180,E1 12344.691,E2 12344.691} C_VEL
LIN {X 0,Y 355.867,Z 936.699,A -85,B 0,C 180,E1 12349.831,E2 12349.831} C_VEL
LIN {X 0,Y 354.871,Z 940.337,A -85,B 0,C 180,E1 12355.166,E2 12355.166} C_VEL
LIN {X 0,Y 355.126,Z 939.772,A -85,B 0,C 180,E1 12360.658,E2 12360.658} C_VEL
LIN {X 0,Y 356.426,Z 934.443,A -85,B 0,C 180,E1 12366.497,E2 12366.497} C_VEL
LIN {X 0,Y 358.409,Z 923.929,A -85,B 0,C 180,E1 12372.35,E2 12372.35} C_VEL
LIN {X 0,Y 362.256,Z 908.115,A -85,B 0,C 180,E1 12377.977,E2 12377.977} C_VEL
LIN {X 0,Y 367.557,Z 888.086,A -85,B 0,C 180,E1 12382.967,E2 12382.967} C_VEL
LIN {X 0,Y 374.455,Z 862.421,A -85,B 0,C 180,E1 12387.573,E2 12387.573} C_VEL
LIN {X 0,Y 381.883,Z 832.269,A -85,B 0,C 180,E1 12391.436,E2 12391.436} C_VEL
LIN {X 0,Y 388.625,Z 799.963,A -85,B 0,C 180,E1 12394.375,E2 12394.375} C_VEL
LIN {X 0,Y 391.613,Z 781.05,A -85,B 0,C 180,E1 12395.706,E2 12395.706} C_VEL
LIN {X 0,Y 380.999,Z 750.588,A -85,B 0,C 180,E1 12399.52,E2 12399.52} C_VEL
LIN {X 0,Y 367.415,Z 724.639,A -85,B 0,C 180,E1 12403.315,E2 12403.315} C_VEL
LIN {X 0,Y 356.928,Z 708.46,A -85,B 0,C 180,E1 12406.224,E2 12406.224} C_VEL
LIN {X 0,Y 354.374,Z 703.793,A -85,B 0,C 180,E1 12407.028,E2 12407.028} C_VEL
LIN {X 0,Y 354.301,Z 702.53,A -85,B 0,C 180,E1 12407.259,E2 12407.259} C_VEL
LIN {X 0,Y 354.678,Z 702.53,A -85,B 0,C 180,E1 12415.139,E2 12415.139} C_VEL
LIN {X 0,Y 354.944,Z 702.53,A -85,B 0,C 180,E1 12422.456,E2 12422.456} C_VEL
LIN {X 0,Y 354.311,Z 702.53,A -85,B 0,C 180,E1 12429.826,E2 12429.826} C_VEL
LIN {X 0,Y 353.926,Z 702.53,A -85,B 0,C 180,E1 12437.381,E2 12437.381} C_VEL
LIN {X 0,Y 353.56,Z 702.53,A -85,B 0,C 180,E1 12445.28,E2 12445.28} C_VEL
LIN {X 0,Y 353.307,Z 702.53,A -85,B 0,C 180,E1 12453.742,E2 12453.742} C_VEL
LIN {X 0,Y 356.048,Z 708.535,A -85,B 0,C 180,E1 12454.83,E2 12454.83} C_VEL
LIN {X 0,Y 358.703,Z 712.205,A -85,B 0,C 180,E1 12455.586,E2 12455.586} C_VEL
LIN {X 0,Y 371.569,Z 731.613,A -85,B 0,C 180,E1 12458.902,E2 12458.902} C_VEL
LIN {X 0,Y 387.203,Z 760.676,A -85,B 0,C 180,E1 12462.575,E2 12462.575} C_VEL
LIN {X 0,Y 397.57,Z 787.562,A -85,B 0,C 180,E1 12465.368,E2 12465.368} C_VEL
LIN {X 0,Y 391.874,Z 824.822,A -85,B 0,C 180,E1 12467.264,E2 12467.264} C_VEL
LIN {X 0,Y 384.608,Z 861.427,A -85,B 0,C 180,E1 12470.052,E2 12470.052} C_VEL
LIN {X 0,Y 376.628,Z 895.882,A -85,B 0,C 180,E1 12473.773,E2 12473.773} C_VEL
LIN {X 0,Y 368.966,Z 927.057,A -85,B 0,C 180,E1 12478.415,E2 12478.415} C_VEL
LIN {X 0,Y 362.652,Z 953.761,A -85,B 0,C 180,E1 12483.873,E2 12483.873} C_VEL
LIN {X 0,Y 358.468,Z 974.481,A -85,B 0,C 180,E1 12489.678,E2 12489.678} C_VEL
LIN {X 0,Y 356.135,Z 989.934,A -85,B 0,C 180,E1 12495.823,E2 12495.823} C_VEL
LIN {X 0,Y 355.402,Z 999.115,A -85,B 0,C 180,E1 12501.453,E2 12501.453} C_VEL
LIN {X 0,Y 355.305,Z 1003.903,A -85,B 0,C 180,E1 12507.566,E2 12507.566} C_VEL
LIN {X 0,Y 355.329,Z 1003.964,A -85,B 0,C 180,E1 12512.434,E2 12512.434} C_VEL
LIN {X 0,Y 355.385,Z 999.339,A -85,B 0,C 180,E1 12518.546,E2 12518.546} C_VEL
LIN {X 0,Y 355.686,Z 995.484,A -85,B 0,C 180,E1 12521.289,E2 12521.289} C_VEL
LIN {X 0,Y 353.481,Z 991.971,A -85,B 0,C 180,E1 12523.3,E2 12523.3} C_VEL
LIN {X 0,Y 348.885,Z 985.807,A -85,B 0,C 180,E1 12526.297,E2 12526.297} C_VEL
LIN {X 0,Y 348.915,Z 985.048,A -85,B 0,C 180,E1 12526.638,E2 12526.638} C_VEL
LIN {X 0,Y 351.939,Z 968.337,A -85,B 0,C 180,E1 12532.699,E2 12532.699} C_VEL
LIN {X 0,Y 357.011,Z 946.419,A -85,B 0,C 180,E1 12538.393,E2 12538.393} C_VEL
LIN {X 0,Y 364.199,Z 918.596,A -85,B 0,C 180,E1 12543.673,E2 12543.673} C_VEL
LIN {X 0,Y 372.167,Z 887.272,A -85,B 0,C 180,E1 12547.993,E2 12547.993} C_VEL
LIN {X 0,Y 380.257,Z 852.242,A -85,B 0,C 180,E1 12551.467,E2 12551.467} C_VEL
LIN {X 0,Y 387.226,Z 815.745,A -85,B 0,C 180,E1 12553.988,E2 12553.988} C_VEL
LIN {X 0,Y 390.598,Z 788.741,A -85,B 0,C 180,E1 12555.355,E2 12555.355} C_VEL
LIN {X 0,Y 375.825,Z 754.861,A -85,B 0,C 180,E1 12558.974,E2 12558.974} C_VEL
LIN {X 0,Y 354.611,Z 718.796,A -85,B 0,C 180,E1 12563.537,E2 12563.537} C_VEL
LIN {X 0,Y 345.564,Z 704.117,A -85,B 0,C 180,E1 12565.703,E2 12565.703} C_VEL
LIN {X 0,Y 345.401,Z 702.53,A -85,B 0,C 180,E1 12565.99,E2 12565.99} C_VEL
LIN {X 0,Y 345.658,Z 702.53,A -85,B 0,C 180,E1 12574.099,E2 12574.099} C_VEL
LIN {X 0,Y 346.024,Z 702.53,A -85,B 0,C 180,E1 12582.209,E2 12582.209} C_VEL
LIN {X 0,Y 346.439,Z 702.53,A -85,B 0,C 180,E1 12589.948,E2 12589.948} C_VEL
LIN {X 0,Y 346.953,Z 702.53,A -85,B 0,C 180,E1 12597.488,E2 12597.488} C_VEL
LIN {X 0,Y 347.041,Z 702.53,A -85,B 0,C 180,E1 12602.472,E2 12602.472} C_VEL
LIN {X 0,Y 346.438,Z 702.53,A -85,B 0,C 180,E1 12610.011,E2 12610.011} C_VEL
LIN {X 0,Y 346.023,Z 702.53,A -85,B 0,C 180,E1 12617.749,E2 12617.749} C_VEL
LIN {X 0,Y 345.633,Z 702.53,A -85,B 0,C 180,E1 12625.858,E2 12625.858} C_VEL
LIN {X 0,Y 345.412,Z 702.53,A -85,B 0,C 180,E1 12633.895,E2 12633.895} C_VEL
LIN {X 0,Y 345.204,Z 702.53,A -85,B 0,C 180,E1 12640.935,E2 12640.935} C_VEL
LIN {X 0,Y 345.166,Z 702.53,A -85,B 0,C 180,E1 12647.961,E2 12647.961} C_VEL
LIN {X 0,Y 345.407,Z 702.53,A -85,B 0,C 180,E1 12655.393,E2 12655.393} C_VEL
LIN {X 0,Y 345.536,Z 702.53,A -85,B 0,C 180,E1 12661.289,E2 12661.289} C_VEL
LIN {X 0,Y 345.959,Z 703.313,A -85,B 0,C 180,E1 12667.824,E2 12667.824} C_VEL
LIN {X 0,Y 348.824,Z 708.657,A -85,B 0,C 180,E1 12668.537,E2 12668.537} C_VEL
LIN {X 0,Y 367.091,Z 740.291,A -85,B 0,C 180,E1 12672.902,E2 12672.902} C_VEL
LIN {X 0,Y 379.857,Z 771.048,A -85,B 0,C 180,E1 12676.677,E2 12676.677} C_VEL
LIN {X 0,Y 383.033,Z 783.636,A -85,B 0,C 180,E1 12678.098,E2 12678.098} C_VEL
LIN {X 0,Y 376.614,Z 818.029,A -85,B 0,C 180,E1 12680.778,E2 12680.778} C_VEL
LIN {X 0,Y 369.44,Z 849.474,A -85,B 0,C 180,E1 12684.286,E2 12684.286} C_VEL
LIN {X 0,Y 362.035,Z 878.298,A -85,B 0,C 180,E1 12688.822,E2 12688.822} C_VEL
LIN {X 0,Y 355.921,Z 901.118,A -85,B 0,C 180,E1 12693.851,E2 12693.851} C_VEL
LIN {X 0,Y 351.603,Z 918.916,A -85,B 0,C 180,E1 12699.409,E2 12699.409} C_VEL
LIN {X 0,Y 348.89,Z 932.152,A -85,B 0,C 180,E1 12705.684,E2 12705.684} C_VEL
LIN {X 0,Y 347.568,Z 939.124,A -85,B 0,C 180,E1 12711.584,E2 12711.584} C_VEL
LIN {X 0,Y 346.946,Z 941.152,A -85,B 0,C 180,E1 12715.782,E2 12715.782} C_VEL
LIN {X 0,Y 347.359,Z 940.106,A -85,B 0,C 180,E1 12721.421,E2 12721.421} C_VEL
LIN {X 0,Y 348.75,Z 934.381,A -85,B 0,C 180,E1 12727.285,E2 12727.285} C_VEL
LIN {X 0,Y 351.185,Z 923.009,A -85,B 0,C 180,E1 12733.434,E2 12733.434} C_VEL
LIN {X 0,Y 355.365,Z 907.272,A -85,B 0,C 180,E1 12738.935,E2 12738.935} C_VEL
LIN {X 0,Y 361.501,Z 885.481,A -85,B 0,C 180,E1 12744.272,E2 12744.272} C_VEL
LIN {X 0,Y 368.969,Z 858.697,A -85,B 0,C 180,E1 12748.9,E2 12748.9} C_VEL
LIN {X 0,Y 376.478,Z 829.268,A -85,B 0,C 180,E1 12752.553,E2 12752.553} C_VEL
LIN {X 0,Y 383.508,Z 796.452,A -85,B 0,C 180,E1 12755.447,E2 12755.447} C_VEL
LIN {X 0,Y 385.441,Z 783.88,A -85,B 0,C 180,E1 12756.355,E2 12756.355} C_VEL
LIN {X 0,Y 375.265,Z 753.985,A -85,B 0,C 180,E1 12760.267,E2 12760.267} C_VEL
LIN {X 0,Y 361.619,Z 727.177,A -85,B 0,C 180,E1 12764.41,E2 12764.41} C_VEL
LIN {X 0,Y 349.582,Z 708.826,A -85,B 0,C 180,E1 12768.044,E2 12768.044} C_VEL
LIN {X 0,Y 346.522,Z 703.617,A -85,B 0,C 180,E1 12769.107,E2 12769.107} C_VEL
LIN {X 0,Y 346.454,Z 702.53,A -85,B 0,C 180,E1 12769.573,E2 12769.573} C_VEL
LIN {X 0,Y 346.932,Z 702.53,A -85,B 0,C 180,E1 12777.528,E2 12777.528} C_VEL
LIN {X 0,Y 347.049,Z 702.53,A -85,B 0,C 180,E1 12782.512,E2 12782.512} C_VEL
LIN {X 0,Y 346.382,Z 702.53,A -85,B 0,C 180,E1 12790.054,E2 12790.054} C_VEL
LIN {X 0,Y 345.965,Z 702.53,A -85,B 0,C 180,E1 12797.794,E2 12797.794} C_VEL
LIN {X 0,Y 345.62,Z 702.53,A -85,B 0,C 180,E1 12805.904,E2 12805.904} C_VEL
LIN {X 0,Y 345.374,Z 702.53,A -85,B 0,C 180,E1 12811.759,E2 12811.759} C_VEL
LIN {X 0,Y 347.384,Z 707.827,A -85,B 0,C 180,E1 12812.567,E2 12812.567} C_VEL
LIN {X 0,Y 350.477,Z 711.495,A -85,B 0,C 180,E1 12813.546,E2 12813.546} C_VEL
LIN {X 0,Y 363.485,Z 730.612,A -85,B 0,C 180,E1 12817.259,E2 12817.259} C_VEL
LIN {X 0,Y 378.782,Z 758.015,A -85,B 0,C 180,E1 12821.111,E2 12821.111} C_VEL
LIN {X 0,Y 391.231,Z 789.394,A -85,B 0,C 180,E1 12824.62,E2 12824.62} C_VEL
LIN {X 0,Y 384.84,Z 830.401,A -85,B 0,C 180,E1 12826.872,E2 12826.872} C_VEL
LIN {X 0,Y 376.717,Z 867.775,A -85,B 0,C 180,E1 12829.945,E2 12829.945} C_VEL
LIN {X 0,Y 368.57,Z 900.647,A -85,B 0,C 180,E1 12833.764,E2 12833.764} C_VEL
LIN {X 0,Y 360.751,Z 930.702,A -85,B 0,C 180,E1 12838.553,E2 12838.553} C_VEL
LIN {X 0,Y 354.64,Z 955.501,A -85,B 0,C 180,E1 12843.922,E2 12843.922} C_VEL
LIN {X 0,Y 350.423,Z 975.55,A -85,B 0,C 180,E1 12849.848,E2 12849.848} C_VEL
LIN {X 0,Y 348.145,Z 990.56,A -85,B 0,C 180,E1 12856.208,E2 12856.208} C_VEL
LIN {X 0,Y 347.552,Z 998.393,A -85,B 0,C 180,E1 12861.259,E2 12861.259} C_VEL
LIN {X 0,Y 347.442,Z 1003.195,A -85,B 0,C 180,E1 12867.51,E2 12867.51} C_VEL
LIN {X 0,Y 347.457,Z 1003.235,A -85,B 0,C 180,E1 12872.545,E2 12872.545} C_VEL
LIN {X 0,Y 347.502,Z 998.621,A -85,B 0,C 180,E1 12878.742,E2 12878.742} C_VEL
LIN {X 0,Y 348.466,Z 988.507,A -85,B 0,C 180,E1 12885.06,E2 12885.06} C_VEL
LIN {X 0,Y 348.915,Z 985.048,A -85,B 0,C 180,E1 12886.638,E2 12886.638} C_VEL
LIN {X 0,Y 347.157,Z 980.437,A -85,B 0,C 180,E1 12888.644,E2 12888.644} C_VEL
LIN {X 0,Y 343.319,Z 972.582,A -85,B 0,C 180,E1 12891.606,E2 12891.606} C_VEL
LIN {X 0,Y 343.442,Z 971.583,A -85,B 0,C 180,E1 12891.933,E2 12891.933} C_VEL
LIN {X 0,Y 348.757,Z 949.431,A -85,B 0,C 180,E1 12898.136,E2 12898.136} C_VEL
LIN {X 0,Y 355.734,Z 923.152,A -85,B 0,C 180,E1 12903.467,E2 12903.467} C_VEL
LIN {X 0,Y 364.029,Z 892.379,A -85,B 0,C 180,E1 12908.023,E2 12908.023} C_VEL
LIN {X 0,Y 372.296,Z 859.265,A -85,B 0,C 180,E1 12911.564,E2 12911.564} C_VEL
LIN {X 0,Y 379.771,Z 823.095,A -85,B 0,C 180,E1 12914.301,E2 12914.301} C_VEL
LIN {X 0,Y 384.376,Z 791.568,A -85,B 0,C 180,E1 12915.996,E2 12915.996} C_VEL
LIN {X 0,Y 369.955,Z 758.137,A -85,B 0,C 180,E1 12919.727,E2 12919.727} C_VEL
LIN {X 0,Y 350.082,Z 723.886,A -85,B 0,C 180,E1 12924.21,E2 12924.21} C_VEL
LIN {X 0,Y 337.591,Z 703.805,A -85,B 0,C 180,E1 12927.338,E2 12927.338} C_VEL
LIN {X 0,Y 337.491,Z 702.53,A -85,B 0,C 180,E1 12927.535,E2 12927.535} C_VEL
LIN {X 0,Y 337.642,Z 702.53,A -85,B 0,C 180,E1 12933.437,E2 12933.437} C_VEL
LIN {X 0,Y 337.989,Z 702.53,A -85,B 0,C 180,E1 12939.65,E2 12939.65} C_VEL
LIN {X 0,Y 338.389,Z 702.53,A -85,B 0,C 180,E1 12947.098,E2 12947.098} C_VEL
LIN {X 0,Y 338.865,Z 702.53,A -85,B 0,C 180,E1 12954.871,E2 12954.871} C_VEL
LIN {X 0,Y 339.171,Z 702.53,A -85,B 0,C 180,E1 12959.98,E2 12959.98} C_VEL
LIN {X 0,Y 338.724,Z 702.53,A -85,B 0,C 180,E1 12967.658,E2 12967.658} C_VEL
LIN {X 0,Y 338.218,Z 702.53,A -85,B 0,C 180,E1 12975.502,E2 12975.502} C_VEL
LIN {X 0,Y 337.887,Z 702.53,A -85,B 0,C 180,E1 12980.906,E2 12980.906} C_VEL
LIN {X 0,Y 337.612,Z 702.53,A -85,B 0,C 180,E1 12986.628,E2 12986.628} C_VEL
LIN {X 0,Y 337.479,Z 702.53,A -85,B 0,C 180,E1 12992.418,E2 12992.418} C_VEL
LIN {X 0,Y 337.282,Z 702.53,A -85,B 0,C 180,E1 13000.484,E2 13000.484} C_VEL
LIN {X 0,Y 337.275,Z 702.53,A -85,B 0,C 180,E1 13007.846,E2 13007.846} C_VEL
LIN {X 0,Y 337.353,Z 702.53,A -85,B 0,C 180,E1 13014.444,E2 13014.444} C_VEL
LIN {X 0,Y 337.6,Z 702.53,A -85,B 0,C 180,E1 13020.549,E2 13020.549} C_VEL
LIN {X 0,Y 337.905,Z 703.25,A -85,B 0,C 180,E1 13026.233,E2 13026.233} C_VEL
LIN {X 0,Y 340.894,Z 708.694,A -85,B 0,C 180,E1 13027.02,E2 13027.02} C_VEL
LIN {X 0,Y 359.037,Z 739.432,A -85,B 0,C 180,E1 13031.57,E2 13031.57} C_VEL
LIN {X 0,Y 371.677,Z 768.564,A -85,B 0,C 180,E1 13035.363,E2 13035.363} C_VEL
LIN {X 0,Y 376.711,Z 785.425,A -85,B 0,C 180,E1 13037.43,E2 13037.43} C_VEL
LIN {X 0,Y 369.981,Z 819.752,A -85,B 0,C 180,E1 13040.166,E2 13040.166} C_VEL
LIN {X 0,Y 362.325,Z 852.006,A -85,B 0,C 180,E1 13043.874,E2 13043.874} C_VEL
LIN {X 0,Y 354.775,Z 879.823,A -85,B 0,C 180,E1 13048.399,E2 13048.399} C_VEL
LIN {X 0,Y 348.334,Z 902.682,A -85,B 0,C 180,E1 13053.588,E2 13053.588} C_VEL
LIN {X 0,Y 343.797,Z 920.554,A -85,B 0,C 180,E1 13059.383,E2 13059.383} C_VEL
LIN {X 0,Y 341.147,Z 932.773,A -85,B 0,C 180,E1 13065.391,E2 13065.391} C_VEL
LIN {X 0,Y 339.779,Z 939.662,A -85,B 0,C 180,E1 13071.24,E2 13071.24} C_VEL
LIN {X 0,Y 339.012,Z 942.051,A -85,B 0,C 180,E1 13077.167,E2 13077.167} C_VEL
LIN {X 0,Y 340.018,Z 939.236,A -85,B 0,C 180,E1 13083.78,E2 13083.78} C_VEL
LIN {X 0,Y 341.778,Z 931.331,A -85,B 0,C 180,E1 13090.027,E2 13090.027} C_VEL
LIN {X 0,Y 345.106,Z 918.305,A -85,B 0,C 180,E1 13096.034,E2 13096.034} C_VEL
LIN {X 0,Y 350.683,Z 898.842,A -85,B 0,C 180,E1 13101.993,E2 13101.993} C_VEL
LIN {X 0,Y 357.72,Z 875.549,A -85,B 0,C 180,E1 13106.963,E2 13106.963} C_VEL
LIN {X 0,Y 365.46,Z 848.462,A -85,B 0,C 180,E1 13111.133,E2 13111.133} C_VEL
LIN {X 0,Y 373.531,Z 816.376,A -85,B 0,C 180,E1 13114.666,E2 13114.666} C_VEL
LIN {X 0,Y 379.212,Z 786.513,A -85,B 0,C 180,E1 13117.042,E2 13117.042} C_VEL
LIN {X 0,Y 369.629,Z 757.364,A -85,B 0,C 180,E1 13121.039,E2 13121.039} C_VEL
LIN {X 0,Y 357.184,Z 732.334,A -85,B 0,C 180,E1 13125.13,E2 13125.13} C_VEL
LIN {X 0,Y 346.116,Z 715.11,A -85,B 0,C 180,E1 13128.709,E2 13128.709} C_VEL
LIN {X 0,Y 342.015,Z 709.035,A -85,B 0,C 180,E1 13130.179,E2 13130.179} C_VEL
LIN {X 0,Y 338.744,Z 704.055,A -85,B 0,C 180,E1 13131.456,E2 13131.456} C_VEL
LIN {X 0,Y 338.604,Z 702.53,A -85,B 0,C 180,E1 13131.695,E2 13131.695} C_VEL
LIN {X 0,Y 339.018,Z 702.53,A -85,B 0,C 180,E1 13137.47,E2 13137.47} C_VEL
LIN {X 0,Y 339.13,Z 702.53,A -85,B 0,C 180,E1 13142.57,E2 13142.57} C_VEL
LIN {X 0,Y 338.443,Z 702.53,A -85,B 0,C 180,E1 13150.292,E2 13150.292} C_VEL
LIN {X 0,Y 337.996,Z 702.53,A -85,B 0,C 180,E1 13158.229,E2 13158.229} C_VEL
LIN {X 0,Y 337.793,Z 702.53,A -85,B 0,C 180,E1 13163.723,E2 13163.723} C_VEL
LIN {X 0,Y 337.486,Z 702.581,A -85,B 0,C 180,E1 13169.294,E2 13169.294} C_VEL
LIN {X 0,Y 339.338,Z 707.649,A -85,B 0,C 180,E1 13170.153,E2 13170.153} C_VEL
LIN {X 0,Y 342.71,Z 711.39,A -85,B 0,C 180,E1 13171.376,E2 13171.376} C_VEL
LIN {X 0,Y 356.237,Z 730.952,A -85,B 0,C 180,E1 13175.677,E2 13175.677} C_VEL
LIN {X 0,Y 370.635,Z 755.907,A -85,B 0,C 180,E1 13179.591,E2 13179.591} C_VEL
LIN {X 0,Y 383.017,Z 785.65,A -85,B 0,C 180,E1 13183.216,E2 13183.216} C_VEL
LIN {X 0,Y 385.129,Z 794.042,A -85,B 0,C 180,E1 13184.05,E2 13184.05} C_VEL
LIN {X 0,Y 378.484,Z 831.837,A -85,B 0,C 180,E1 13186.2,E2 13186.2} C_VEL
LIN {X 0,Y 370.131,Z 868.446,A -85,B 0,C 180,E1 13189.283,E2 13189.283} C_VEL
LIN {X 0,Y 361.411,Z 901.829,A -85,B 0,C 180,E1 13193.272,E2 13193.272} C_VEL
LIN {X 0,Y 353.371,Z 931.192,A -85,B 0,C 180,E1 13198.1,E2 13198.1} C_VEL
LIN {X 0,Y 346.819,Z 956.558,A -85,B 0,C 180,E1 13203.795,E2 13203.795} C_VEL
LIN {X 0,Y 342.381,Z 976.621,A -85,B 0,C 180,E1 13210.027,E2 13210.027} C_VEL
LIN {X 0,Y 340.201,Z 991.046,A -85,B 0,C 180,E1 13216.533,E2 13216.533} C_VEL
LIN {X 0,Y 339.584,Z 998.995,A -85,B 0,C 180,E1 13222.339,E2 13222.339} C_VEL
LIN {X 0,Y 339.559,Z 1002.487,A -85,B 0,C 180,E1 13227.453,E2 13227.453} C_VEL
LIN {X 0,Y 339.584,Z 1002.551,A -85,B 0,C 180,E1 13232.547,E2 13232.547} C_VEL
LIN {X 0,Y 339.651,Z 997.903,A -85,B 0,C 180,E1 13238.945,E2 13238.945} C_VEL
LIN {X 0,Y 340.654,Z 987.766,A -85,B 0,C 180,E1 13245.413,E2 13245.413} C_VEL
LIN {X 0,Y 343.442,Z 971.583,A -85,B 0,C 180,E1 13251.933,E2 13251.933} C_VEL
LIN {X 0,Y 341.343,Z 963.737,A -85,B 0,C 180,E1 13254.538,E2 13254.538} C_VEL
LIN {X 0,Y 339.678,Z 955.187,A -85,B 0,C 180,E1 13257.112,E2 13257.112} C_VEL
LIN {X 0,Y 346.449,Z 930.822,A -85,B 0,C 180,E1 13262.616,E2 13262.616} C_VEL
LIN {X 0,Y 354.672,Z 901.65,A -85,B 0,C 180,E1 13267.452,E2 13267.452} C_VEL
LIN {X 0,Y 363.591,Z 868.485,A -85,B 0,C 180,E1 13271.411,E2 13271.411} C_VEL
LIN {X 0,Y 372.022,Z 831.505,A -85,B 0,C 180,E1 13274.523,E2 13274.523} C_VEL
LIN {X 0,Y 378.254,Z 794.746,A -85,B 0,C 180,E1 13276.619,E2 13276.619} C_VEL
LIN {X 0,Y 364.373,Z 761.9,A -85,B 0,C 180,E1 13280.437,E2 13280.437} C_VEL
LIN {X 0,Y 344.504,Z 726.929,A -85,B 0,C 180,E1 13285.179,E2 13285.179} C_VEL
LIN {X 0,Y 331.621,Z 707.798,A -85,B 0,C 180,E1 13288.493,E2 13288.493} C_VEL
LIN {X 0,Y 329.59,Z 702.53,A -85,B 0,C 180,E1 13289.159,E2 13289.159} C_VEL
LIN {X 0,Y 329.913,Z 702.53,A -85,B 0,C 180,E1 13296.177,E2 13296.177} C_VEL
LIN {X 0,Y 330.268,Z 702.53,A -85,B 0,C 180,E1 13304.071,E2 13304.071} C_VEL
LIN {X 0,Y 330.735,Z 702.53,A -85,B 0,C 180,E1 13312.113,E2 13312.113} C_VEL
LIN {X 0,Y 331.286,Z 702.53,A -85,B 0,C 180,E1 13319.979,E2 13319.979} C_VEL
LIN {X 0,Y 330.782,Z 702.53,A -85,B 0,C 180,E1 13327.843,E2 13327.843} C_VEL
LIN {X 0,Y 330.245,Z 702.53,A -85,B 0,C 180,E1 13335.886,E2 13335.886} C_VEL
LIN {X 0,Y 329.782,Z 702.53,A -85,B 0,C 180,E1 13344.29,E2 13344.29} C_VEL
LIN {X 0,Y 329.556,Z 702.53,A -85,B 0,C 180,E1 13350.212,E2 13350.212} C_VEL
LIN {X 0,Y 329.436,Z 702.53,A -85,B 0,C 180,E1 13356.511,E2 13356.511} C_VEL
LIN {X 0,Y 329.345,Z 702.53,A -85,B 0,C 180,E1 13363.374,E2 13363.374} C_VEL
LIN {X 0,Y 329.366,Z 702.53,A -85,B 0,C 180,E1 13371.107,E2 13371.107} C_VEL
LIN {X 0,Y 329.456,Z 702.53,A -85,B 0,C 180,E1 13376.658,E2 13376.658} C_VEL
LIN {X 0,Y 329.828,Z 702.53,A -85,B 0,C 180,E1 13384.236,E2 13384.236} C_VEL
LIN {X 0,Y 329.93,Z 703.618,A -85,B 0,C 180,E1 13384.551,E2 13384.551} C_VEL
LIN {X 0,Y 333.144,Z 708.927,A -85,B 0,C 180,E1 13385.445,E2 13385.445} C_VEL
LIN {X 0,Y 351.02,Z 738.62,A -85,B 0,C 180,E1 13390.156,E2 13390.156} C_VEL
LIN {X 0,Y 363.978,Z 767.339,A -85,B 0,C 180,E1 13394.145,E2 13394.145} C_VEL
LIN {X 0,Y 370.131,Z 788.962,A -85,B 0,C 180,E1 13396.857,E2 13396.857} C_VEL
LIN {X 0,Y 362.724,Z 824.384,A -85,B 0,C 180,E1 13399.816,E2 13399.816} C_VEL
LIN {X 0,Y 354.866,Z 855.435,A -85,B 0,C 180,E1 13403.591,E2 13403.591} C_VEL
LIN {X 0,Y 347.581,Z 881.09,A -85,B 0,C 180,E1 13407.906,E2 13407.906} C_VEL
LIN {X 0,Y 340.852,Z 903.96,A -85,B 0,C 180,E1 13413.238,E2 13413.238} C_VEL
LIN {X 0,Y 336.08,Z 921.675,A -85,B 0,C 180,E1 13419.17,E2 13419.17} C_VEL
LIN {X 0,Y 333.213,Z 934.374,A -85,B 0,C 180,E1 13425.767,E2 13425.767} C_VEL
LIN {X 0,Y 331.88,Z 940.503,A -85,B 0,C 180,E1 13431.331,E2 13431.331} C_VEL
LIN {X 0,Y 331.157,Z 942.768,A -85,B 0,C 180,E1 13437.109,E2 13437.109} C_VEL
LIN {X 0,Y 331.977,Z 940.713,A -85,B 0,C 180,E1 13443.057,E2 13443.057} C_VEL
LIN {X 0,Y 333.718,Z 933.832,A -85,B 0,C 180,E1 13449.277,E2 13449.277} C_VEL
LIN {X 0,Y 337.066,Z 920.965,A -85,B 0,C 180,E1 13455.751,E2 13455.751} C_VEL
LIN {X 0,Y 342.735,Z 902.369,A -85,B 0,C 180,E1 13461.85,E2 13461.85} C_VEL
LIN {X 0,Y 350.111,Z 879.174,A -85,B 0,C 180,E1 13467.124,E2 13467.124} C_VEL
LIN {X 0,Y 358.442,Z 851.573,A -85,B 0,C 180,E1 13471.571,E2 13471.571} C_VEL
LIN {X 0,Y 366.617,Z 820.923,A -85,B 0,C 180,E1 13475.095,E2 13475.095} C_VEL
LIN {X 0,Y 373.056,Z 789.322,A -85,B 0,C 180,E1 13477.74,E2 13477.74} C_VEL
LIN {X 0,Y 364.078,Z 760.862,A -85,B 0,C 180,E1 13481.829,E2 13481.829} C_VEL
LIN {X 0,Y 351.394,Z 734.566,A -85,B 0,C 180,E1 13486.362,E2 13486.362} C_VEL
LIN {X 0,Y 339.34,Z 715.999,A -85,B 0,C 180,E1 13490.666,E2 13490.666} C_VEL
LIN {X 0,Y 334.444,Z 709.2,A -85,B 0,C 180,E1 13492.665,E2 13492.665} C_VEL
LIN {X 0,Y 331.089,Z 704.419,A -85,B 0,C 180,E1 13494.218,E2 13494.218} C_VEL
LIN {X 0,Y 330.883,Z 702.53,A -85,B 0,C 180,E1 13494.461,E2 13494.461} C_VEL
LIN {X 0,Y 331.29,Z 702.53,A -85,B 0,C 180,E1 13500.021,E2 13500.021} C_VEL
LIN {X 0,Y 330.927,Z 702.53,A -85,B 0,C 180,E1 13505.252,E2 13505.252} C_VEL
LIN {X 0,Y 330.382,Z 702.53,A -85,B 0,C 180,E1 13513.22,E2 13513.22} C_VEL
LIN {X 0,Y 329.914,Z 702.53,A -85,B 0,C 180,E1 13521.481,E2 13521.481} C_VEL
LIN {X 0,Y 329.715,Z 702.53,A -85,B 0,C 180,E1 13526.32,E2 13526.32} C_VEL
LIN {X 0,Y 331.634,Z 707.791,A -85,B 0,C 180,E1 13527.424,E2 13527.424} C_VEL
LIN {X 0,Y 334.947,Z 711.079,A -85,B 0,C 180,E1 13528.829,E2 13528.829} C_VEL
LIN {X 0,Y 345.87,Z 726.984,A -85,B 0,C 180,E1 13532.93,E2 13532.93} C_VEL
LIN {X 0,Y 358.158,Z 745.812,A -85,B 0,C 180,E1 13536.669,E2 13536.669} C_VEL
LIN {X 0,Y 371.535,Z 773.389,A -85,B 0,C 180,E1 13540.639,E2 13540.639} C_VEL
LIN {X 0,Y 379.192,Z 795.839,A -85,B 0,C 180,E1 13543.31,E2 13543.31} C_VEL
LIN {X 0,Y 372.416,Z 832.323,A -85,B 0,C 180,E1 13545.43,E2 13545.43} C_VEL
LIN {X 0,Y 363.992,Z 867.642,A -85,B 0,C 180,E1 13548.446,E2 13548.446} C_VEL
LIN {X 0,Y 355.209,Z 899.886,A -85,B 0,C 180,E1 13552.316,E2 13552.316} C_VEL
LIN {X 0,Y 346.866,Z 928.747,A -85,B 0,C 180,E1 13557.056,E2 13557.056} C_VEL
LIN {X 0,Y 340.002,Z 953.556,A -85,B 0,C 180,E1 13562.598,E2 13562.598} C_VEL
LIN {X 0,Y 335.097,Z 974.025,A -85,B 0,C 180,E1 13568.883,E2 13568.883} C_VEL
LIN {X 0,Y 332.547,Z 989.086,A -85,B 0,C 180,E1 13575.547,E2 13575.547} C_VEL
LIN {X 0,Y 331.841,Z 996.949,A -85,B 0,C 180,E1 13580.841,E2 13580.841} C_VEL
LIN {X 0,Y 331.695,Z 1001.78,A -85,B 0,C 180,E1 13587.392,E2 13587.392} C_VEL
LIN {X 0,Y 331.711,Z 1001.843,A -85,B 0,C 180,E1 13592.607,E2 13592.607} C_VEL
LIN {X 0,Y 331.797,Z 997.181,A -85,B 0,C 180,E1 13599.159,E2 13599.159} C_VEL
LIN {X 0,Y 332.842,Z 987.007,A -85,B 0,C 180,E1 13605.784,E2 13605.784} C_VEL
LIN {X 0,Y 335.695,Z 971.479,A -85,B 0,C 180,E1 13612.224,E2 13612.224} C_VEL
LIN {X 0,Y 339.678,Z 955.187,A -85,B 0,C 180,E1 13617.112,E2 13617.112} C_VEL
LIN {X 0,Y 338.482,Z 946.007,A -85,B 0,C 180,E1 13619.627,E2 13619.627} C_VEL
LIN {X 0,Y 337.681,Z 936.164,A -85,B 0,C 180,E1 13622.09,E2 13622.09} C_VEL
LIN {X 0,Y 346.339,Z 907.043,A -85,B 0,C 180,E1 13627.329,E2 13627.329} C_VEL
LIN {X 0,Y 355.933,Z 872.927,A -85,B 0,C 180,E1 13631.689,E2 13631.689} C_VEL
LIN {X 0,Y 364.604,Z 837.47,A -85,B 0,C 180,E1 13634.869,E2 13634.869} C_VEL
LIN {X 0,Y 371.591,Z 800.943,A -85,B 0,C 180,E1 13637.097,E2 13637.097} C_VEL
LIN {X 0,Y 371.438,Z 795.958,A -85,B 0,C 180,E1 13637.469,E2 13637.469} C_VEL
LIN {X 0,Y 358.329,Z 764.647,A -85,B 0,C 180,E1 13641.296,E2 13641.296} C_VEL
LIN {X 0,Y 339.968,Z 732.098,A -85,B 0,C 180,E1 13645.902,E2 13645.902} C_VEL
LIN {X 0,Y 323.966,Z 708.023,A -85,B 0,C 180,E1 13650.247,E2 13650.247} C_VEL
LIN {X 0,Y 321.707,Z 702.53,A -85,B 0,C 180,E1 13651.16,E2 13651.16} C_VEL
LIN {X 0,Y 321.999,Z 702.53,A -85,B 0,C 180,E1 13657.963,E2 13657.963} C_VEL
LIN {X 0,Y 322.483,Z 702.53,A -85,B 0,C 180,E1 13666.45,E2 13666.45} C_VEL
LIN {X 0,Y 323.013,Z 702.53,A -85,B 0,C 180,E1 13674.618,E2 13674.618} C_VEL
LIN {X 0,Y 323.383,Z 702.53,A -85,B 0,C 180,E1 13679.979,E2 13679.979} C_VEL
LIN {X 0,Y 322.84,Z 702.53,A -85,B 0,C 180,E1 13688.037,E2 13688.037} C_VEL
LIN {X 0,Y 322.293,Z 702.53,A -85,B 0,C 180,E1 13696.289,E2 13696.289} C_VEL
LIN {X 0,Y 321.965,Z 702.53,A -85,B 0,C 180,E1 13701.993,E2 13701.993} C_VEL
LIN {X 0,Y 321.693,Z 702.53,A -85,B 0,C 180,E1 13707.943,E2 13707.943} C_VEL
LIN {X 0,Y 321.507,Z 702.53,A -85,B 0,C 180,E1 13714.244,E2 13714.244} C_VEL
LIN {X 0,Y 321.346,Z 702.53,A -85,B 0,C 180,E1 13721.293,E2 13721.293} C_VEL
LIN {X 0,Y 321.322,Z 702.53,A -85,B 0,C 180,E1 13728.892,E2 13728.892} C_VEL
LIN {X 0,Y 321.551,Z 702.53,A -85,B 0,C 180,E1 13735.726,E2 13735.726} C_VEL
LIN {X 0,Y 321.837,Z 702.53,A -85,B 0,C 180,E1 13742.641,E2 13742.641} C_VEL
LIN {X 0,Y 324.095,Z 708.049,A -85,B 0,C 180,E1 13743.406,E2 13743.406} C_VEL
LIN {X 0,Y 334.741,Z 723.794,A -85,B 0,C 180,E1 13746.357,E2 13746.357} C_VEL
LIN {X 0,Y 350.144,Z 751.74,A -85,B 0,C 180,E1 13750.794,E2 13750.794} C_VEL
LIN {X 0,Y 361.133,Z 780.358,A -85,B 0,C 180,E1 13754.779,E2 13754.779} C_VEL
LIN {X 0,Y 363.717,Z 791.553,A -85,B 0,C 180,E1 13756.199,E2 13756.199} C_VEL
LIN {X 0,Y 356.173,Z 825.965,A -85,B 0,C 180,E1 13759.164,E2 13759.164} C_VEL
LIN {X 0,Y 348.029,Z 856.802,A -85,B 0,C 180,E1 13762.996,E2 13762.996} C_VEL
LIN {X 0,Y 340.313,Z 882.677,A -85,B 0,C 180,E1 13767.459,E2 13767.459} C_VEL
LIN {X 0,Y 333.214,Z 905.734,A -85,B 0,C 180,E1 13773.012,E2 13773.012} C_VEL
LIN {X 0,Y 328.57,Z 922.091,A -85,B 0,C 180,E1 13778.65,E2 13778.65} C_VEL
LIN {X 0,Y 325.627,Z 934.105,A -85,B 0,C 180,E1 13784.835,E2 13784.835} C_VEL
LIN {X 0,Y 324.254,Z 940.395,A -85,B 0,C 180,E1 13790.199,E2 13790.199} C_VEL
LIN {X 0,Y 323.386,Z 943.103,A -85,B 0,C 180,E1 13794.833,E2 13794.833} C_VEL
LIN {X 0,Y 323.624,Z 942.728,A -85,B 0,C 180,E1 13800.859,E2 13800.859} C_VEL
LIN {X 0,Y 325.212,Z 937.82,A -85,B 0,C 180,E1 13807.101,E2 13807.101} C_VEL
LIN {X 0,Y 327.878,Z 927.491,A -85,B 0,C 180,E1 13813.659,E2 13813.659} C_VEL
LIN {X 0,Y 332.758,Z 911.949,A -85,B 0,C 180,E1 13819.8,E2 13819.8} C_VEL
LIN {X 0,Y 339.567,Z 891.445,A -85,B 0,C 180,E1 13825.386,E2 13825.386} C_VEL
LIN {X 0,Y 347.762,Z 866.552,A -85,B 0,C 180,E1 13830.21,E2 13830.21} C_VEL
LIN {X 0,Y 356.821,Z 836.437,A -85,B 0,C 180,E1 13834.357,E2 13834.357} C_VEL
LIN {X 0,Y 364.872,Z 804.427,A -85,B 0,C 180,E1 13837.453,E2 13837.453} C_VEL
LIN {X 0,Y 366.961,Z 792.135,A -85,B 0,C 180,E1 13838.462,E2 13838.462} C_VEL
LIN {X 0,Y 358.74,Z 764.8,A -85,B 0,C 180,E1 13842.584,E2 13842.584} C_VEL
LIN {X 0,Y 347.091,Z 739.943,A -85,B 0,C 180,E1 13847.105,E2 13847.105} C_VEL
LIN {X 0,Y 336.433,Z 722.754,A -85,B 0,C 180,E1 13851.245,E2 13851.245} C_VEL
LIN {X 0,Y 331.439,Z 715.808,A -85,B 0,C 180,E1 13853.405,E2 13853.405} C_VEL
LIN {X 0,Y 327.494,Z 709.654,A -85,B 0,C 180,E1 13855.397,E2 13855.397} C_VEL
LIN {X 0,Y 323.606,Z 704.958,A -85,B 0,C 180,E1 13857.6,E2 13857.6} C_VEL
LIN {X 0,Y 323.207,Z 702.53,A -85,B 0,C 180,E1 13858.015,E2 13858.015} C_VEL
LIN {X 0,Y 323.289,Z 702.53,A -85,B 0,C 180,E1 13862.696,E2 13862.696} C_VEL
LIN {X 0,Y 322.595,Z 702.53,A -85,B 0,C 180,E1 13870.804,E2 13870.804} C_VEL
LIN {X 0,Y 322.07,Z 702.53,A -85,B 0,C 180,E1 13879.164,E2 13879.164} C_VEL
LIN {X 0,Y 321.998,Z 703.358,A -85,B 0,C 180,E1 13882.602,E2 13882.602} C_VEL
LIN {X 0,Y 324.683,Z 708.564,A -85,B 0,C 180,E1 13884.421,E2 13884.421} C_VEL
LIN {X 0,Y 327.478,Z 711.016,A -85,B 0,C 180,E1 13885.886,E2 13885.886} C_VEL
LIN {X 0,Y 331.338,Z 716.61,A -85,B 0,C 180,E1 13887.793,E2 13887.793} C_VEL
LIN {X 0,Y 342.26,Z 732.466,A -85,B 0,C 180,E1 13892.145,E2 13892.145} C_VEL
LIN {X 0,Y 354.399,Z 751.793,A -85,B 0,C 180,E1 13896.095,E2 13896.095} C_VEL
LIN {X 0,Y 366.785,Z 778.707,A -85,B 0,C 180,E1 13900.114,E2 13900.114} C_VEL
LIN {X 0,Y 373.007,Z 799.544,A -85,B 0,C 180,E1 13902.627,E2 13902.627} C_VEL
LIN {X 0,Y 365.584,Z 836.485,A -85,B 0,C 180,E1 13904.902,E2 13904.902} C_VEL
LIN {X 0,Y 356.423,Z 872.601,A -85,B 0,C 180,E1 13908.177,E2 13908.177} C_VEL
LIN {X 0,Y 346.782,Z 905.808,A -85,B 0,C 180,E1 13912.467,E2 13912.467} C_VEL
LIN {X 0,Y 338.051,Z 934.475,A -85,B 0,C 180,E1 13917.61,E2 13917.61} C_VEL
LIN {X 0,Y 331.074,Z 958.81,A -85,B 0,C 180,E1 13923.614,E2 13923.614} C_VEL
LIN {X 0,Y 326.698,Z 976.811,A -85,B 0,C 180,E1 13929.731,E2 13929.731} C_VEL
LIN {X 0,Y 324.429,Z 990.652,A -85,B 0,C 180,E1 13936.551,E2 13936.551} C_VEL
LIN {X 0,Y 323.86,Z 997.565,A -85,B 0,C 180,E1 13941.964,E2 13941.964} C_VEL
LIN {X 0,Y 323.811,Z 1001.074,A -85,B 0,C 180,E1 13947.329,E2 13947.329} C_VEL
LIN {X 0,Y 323.827,Z 1001.131,A -85,B 0,C 180,E1 13952.671,E2 13952.671} C_VEL
LIN {X 0,Y 323.918,Z 996.449,A -85,B 0,C 180,E1 13959.384,E2 13959.384} C_VEL
LIN {X 0,Y 325.067,Z 986.249,A -85,B 0,C 180,E1 13966.172,E2 13966.172} C_VEL
LIN {X 0,Y 328.51,Z 969.242,A -85,B 0,C 180,E1 13973.24,E2 13973.24} C_VEL
LIN {X 0,Y 334.087,Z 948.279,A -85,B 0,C 180,E1 13979.321,E2 13979.321} C_VEL
LIN {X 0,Y 337.681,Z 936.164,A -85,B 0,C 180,E1 13982.09,E2 13982.09} C_VEL
LIN {X 0,Y 337.315,Z 925.792,A -85,B 0,C 180,E1 13984.491,E2 13984.491} C_VEL
LIN {X 0,Y 337.162,Z 914.559,A -85,B 0,C 180,E1 13986.78,E2 13986.78} C_VEL
LIN {X 0,Y 346.679,Z 882.845,A -85,B 0,C 180,E1 13991.31,E2 13991.31} C_VEL
LIN {X 0,Y 355.937,Z 848.179,A -85,B 0,C 180,E1 13994.815,E2 13994.815} C_VEL
LIN {X 0,Y 363.619,Z 812.693,A -85,B 0,C 180,E1 13997.301,E2 13997.301} C_VEL
LIN {X 0,Y 365.405,Z 799.355,A -85,B 0,C 180,E1 13998.087,E2 13998.087} C_VEL
LIN {X 0,Y 352.216,Z 767.12,A -85,B 0,C 180,E1 14002.208,E2 14002.208} C_VEL
LIN {X 0,Y 334.719,Z 735.948,A -85,B 0,C 180,E1 14006.848,E2 14006.848} C_VEL
LIN {X 0,Y 316.674,Z 708.574,A -85,B 0,C 180,E1 14012.032,E2 14012.032} C_VEL
LIN {X 0,Y 313.973,Z 703.834,A -85,B 0,C 180,E1 14012.932,E2 14012.932} C_VEL
LIN {X 0,Y 313.861,Z 702.53,A -85,B 0,C 180,E1 14013.311,E2 14013.311} C_VEL
LIN {X 0,Y 314.155,Z 702.53,A -85,B 0,C 180,E1 14020.333,E2 14020.333} C_VEL
LIN {X 0,Y 314.518,Z 702.53,A -85,B 0,C 180,E1 14026.1,E2 14026.1} C_VEL
LIN {X 0,Y 315.092,Z 702.53,A -85,B 0,C 180,E1 14034.483,E2 14034.483} C_VEL
LIN {X 0,Y 315.483,Z 702.53,A -85,B 0,C 180,E1 14039.978,E2 14039.978} C_VEL
LIN {X 0,Y 315.111,Z 702.53,A -85,B 0,C 180,E1 14045.473,E2 14045.473} C_VEL
LIN {X 0,Y 314.546,Z 702.53,A -85,B 0,C 180,E1 14053.853,E2 14053.853} C_VEL
LIN {X 0,Y 314.146,Z 702.53,A -85,B 0,C 180,E1 14059.62,E2 14059.62} C_VEL
LIN {X 0,Y 313.837,Z 702.53,A -85,B 0,C 180,E1 14065.611,E2 14065.611} C_VEL
LIN {X 0,Y 313.621,Z 702.53,A -85,B 0,C 180,E1 14071.922,E2 14071.922} C_VEL
LIN {X 0,Y 313.364,Z 702.53,A -85,B 0,C 180,E1 14079.603,E2 14079.603} C_VEL
LIN {X 0,Y 313.299,Z 702.53,A -85,B 0,C 180,E1 14087.599,E2 14087.599} C_VEL
LIN {X 0,Y 313.544,Z 702.53,A -85,B 0,C 180,E1 14094.845,E2 14094.845} C_VEL
LIN {X 0,Y 313.71,Z 703.154,A -85,B 0,C 180,E1 14100.655,E2 14100.655} C_VEL
LIN {X 0,Y 316.465,Z 708.464,A -85,B 0,C 180,E1 14101.58,E2 14101.58} C_VEL
LIN {X 0,Y 330.298,Z 728.995,A -85,B 0,C 180,E1 14105.659,E2 14105.659} C_VEL
LIN {X 0,Y 345.021,Z 756.721,A -85,B 0,C 180,E1 14110.245,E2 14110.245} C_VEL
LIN {X 0,Y 355.327,Z 784.683,A -85,B 0,C 180,E1 14114.286,E2 14114.286} C_VEL
LIN {X 0,Y 357.431,Z 793.703,A -85,B 0,C 180,E1 14115.489,E2 14115.489} C_VEL
LIN {X 0,Y 349.319,Z 828.858,A -85,B 0,C 180,E1 14118.633,E2 14118.633} C_VEL
LIN {X 0,Y 340.874,Z 859.196,A -85,B 0,C 180,E1 14122.528,E2 14122.528} C_VEL
LIN {X 0,Y 332.461,Z 886.233,A -85,B 0,C 180,E1 14127.399,E2 14127.399} C_VEL
LIN {X 0,Y 325.132,Z 908.886,A -85,B 0,C 180,E1 14133.237,E2 14133.237} C_VEL
LIN {X 0,Y 319.977,Z 926.194,A -85,B 0,C 180,E1 14139.768,E2 14139.768} C_VEL
LIN {X 0,Y 317.334,Z 937.533,A -85,B 0,C 180,E1 14146.578,E2 14146.578} C_VEL
LIN {X 0,Y 315.839,Z 942.801,A -85,B 0,C 180,E1 14152.472,E2 14152.472} C_VEL
LIN {X 0,Y 315.451,Z 944.075,A -85,B 0,C 180,E1 14158.579,E2 14158.579} C_VEL
LIN {X 0,Y 316.706,Z 941.001,A -85,B 0,C 180,E1 14164.874,E2 14164.874} C_VEL
LIN {X 0,Y 318.901,Z 932.915,A -85,B 0,C 180,E1 14171.489,E2 14171.489} C_VEL
LIN {X 0,Y 323.419,Z 918.613,A -85,B 0,C 180,E1 14178.292,E2 14178.292} C_VEL
LIN {X 0,Y 329.945,Z 899.938,A -85,B 0,C 180,E1 14184.172,E2 14184.172} C_VEL
LIN {X 0,Y 338.597,Z 875.315,A -85,B 0,C 180,E1 14189.593,E2 14189.593} C_VEL
LIN {X 0,Y 347.85,Z 847.116,A -85,B 0,C 180,E1 14193.976,E2 14193.976} C_VEL
LIN {X 0,Y 357.134,Z 813.601,A -85,B 0,C 180,E1 14197.61,E2 14197.61} C_VEL
LIN {X 0,Y 361.238,Z 796.165,A -85,B 0,C 180,E1 14199.037,E2 14199.037} C_VEL
LIN {X 0,Y 353.559,Z 769.078,A -85,B 0,C 180,E1 14203.281,E2 14203.281} C_VEL
LIN {X 0,Y 342.979,Z 745.404,A -85,B 0,C 180,E1 14207.816,E2 14207.816} C_VEL
LIN {X 0,Y 333.274,Z 729.056,A -85,B 0,C 180,E1 14211.935,E2 14211.935} C_VEL
LIN {X 0,Y 328.514,Z 722.216,A -85,B 0,C 180,E1 14214.173,E2 14214.173} C_VEL
LIN {X 0,Y 324.923,Z 716.678,A -85,B 0,C 180,E1 14216.093,E2 14216.093} C_VEL
LIN {X 0,Y 321.328,Z 711.265,A -85,B 0,C 180,E1 14218.34,E2 14218.34} C_VEL
LIN {X 0,Y 315.418,Z 704.011,A -85,B 0,C 180,E1 14223.364,E2 14223.364} C_VEL
LIN {X 0,Y 315.147,Z 702.53,A -85,B 0,C 180,E1 14224.14,E2 14224.14} C_VEL
LIN {X 0,Y 314.643,Z 702.53,A -85,B 0,C 180,E1 14231.08,E2 14231.08} C_VEL
LIN {X 0,Y 314.365,Z 703.362,A -85,B 0,C 180,E1 14236.583,E2 14236.583} C_VEL
LIN {X 0,Y 316.696,Z 708.354,A -85,B 0,C 180,E1 14239.502,E2 14239.502} C_VEL
LIN {X 0,Y 320.064,Z 710.891,A -85,B 0,C 180,E1 14242.073,E2 14242.073} C_VEL
LIN {X 0,Y 324.093,Z 716.924,A -85,B 0,C 180,E1 14244.7,E2 14244.7} C_VEL
LIN {X 0,Y 331.101,Z 727.096,A -85,B 0,C 180,E1 14248.262,E2 14248.262} C_VEL
LIN {X 0,Y 342.235,Z 743.262,A -85,B 0,C 180,E1 14252.641,E2 14252.641} C_VEL
LIN {X 0,Y 354.244,Z 765.431,A -85,B 0,C 180,E1 14256.816,E2 14256.816} C_VEL
LIN {X 0,Y 364.6,Z 791.895,A -85,B 0,C 180,E1 14260.646,E2 14260.646} C_VEL
LIN {X 0,Y 367.149,Z 801.667,A -85,B 0,C 180,E1 14261.844,E2 14261.844} C_VEL
LIN {X 0,Y 358.823,Z 840.597,A -85,B 0,C 180,E1 14264.362,E2 14264.362} C_VEL
LIN {X 0,Y 349.187,Z 875.833,A -85,B 0,C 180,E1 14267.73,E2 14267.73} C_VEL
LIN {X 0,Y 339.633,Z 907.053,A -85,B 0,C 180,E1 14271.94,E2 14271.94} C_VEL
LIN {X 0,Y 330.464,Z 935.709,A -85,B 0,C 180,E1 14277.277,E2 14277.277} C_VEL
LIN {X 0,Y 323.388,Z 959.212,A -85,B 0,C 180,E1 14283.312,E2 14283.312} C_VEL
LIN {X 0,Y 318.655,Z 977.703,A -85,B 0,C 180,E1 14289.92,E2 14289.92} C_VEL
LIN {X 0,Y 316.592,Z 989.928,A -85,B 0,C 180,E1 14296.212,E2 14296.212} C_VEL
LIN {X 0,Y 315.981,Z 996.847,A -85,B 0,C 180,E1 14301.762,E2 14301.762} C_VEL
LIN {X 0,Y 315.946,Z 1000.369,A -85,B 0,C 180,E1 14307.262,E2 14307.262} C_VEL
LIN {X 0,Y 315.959,Z 1000.42,A -85,B 0,C 180,E1 14312.737,E2 14312.737} C_VEL
LIN {X 0,Y 316.045,Z 995.717,A -85,B 0,C 180,E1 14319.62,E2 14319.62} C_VEL
LIN {X 0,Y 317.285,Z 985.478,A -85,B 0,C 180,E1 14326.58,E2 14326.58} C_VEL
LIN {X 0,Y 320.674,Z 969.608,A -85,B 0,C 180,E1 14333.409,E2 14333.409} C_VEL
LIN {X 0,Y 326.624,Z 948.365,A -85,B 0,C 180,E1 14339.785,E2 14339.785} C_VEL
LIN {X 0,Y 334.803,Z 921.975,A -85,B 0,C 180,E1 14345.471,E2 14345.471} C_VEL
LIN {X 0,Y 337.162,Z 914.559,A -85,B 0,C 180,E1 14346.78,E2 14346.78} C_VEL
LIN {X 0,Y 337.36,Z 902.832,A -85,B 0,C 180,E1 14348.987,E2 14348.987} C_VEL
LIN {X 0,Y 337.84,Z 890.452,A -85,B 0,C 180,E1 14351.097,E2 14351.097} C_VEL
LIN {X 0,Y 347.569,Z 856.689,A -85,B 0,C 180,E1 14354.871,E2 14354.871} C_VEL
LIN {X 0,Y 356.492,Z 819.086,A -85,B 0,C 180,E1 14357.77,E2 14357.77} C_VEL
LIN {X 0,Y 359.452,Z 802.96,A -85,B 0,C 180,E1 14358.703,E2 14358.703} C_VEL
LIN {X 0,Y 346.858,Z 771.427,A -85,B 0,C 180,E1 14362.891,E2 14362.891} C_VEL
LIN {X 0,Y 330.286,Z 740.888,A -85,B 0,C 180,E1 14367.612,E2 14367.612} C_VEL
LIN {X 0,Y 313.003,Z 714.679,A -85,B 0,C 180,E1 14372.745,E2 14372.745} C_VEL
LIN {X 0,Y 308.656,Z 708.488,A -85,B 0,C 180,E1 14374.192,E2 14374.192} C_VEL
LIN {X 0,Y 306.102,Z 703.969,A -85,B 0,C 180,E1 14375.119,E2 14375.119} C_VEL
LIN {X 0,Y 305.946,Z 702.53,A -85,B 0,C 180,E1 14375.315,E2 14375.315} C_VEL
LIN {X 0,Y 306.353,Z 702.53,A -85,B 0,C 180,E1 14382.79,E2 14382.79} C_VEL
LIN {X 0,Y 306.807,Z 702.53,A -85,B 0,C 180,E1 14389.638,E2 14389.638} C_VEL
LIN {X 0,Y 307.405,Z 702.53,A -85,B 0,C 180,E1 14397.164,E2 14397.164} C_VEL
LIN {X 0,Y 307.456,Z 702.53,A -85,B 0,C 180,E1 14402.79,E2 14402.79} C_VEL
LIN {X 0,Y 306.787,Z 702.53,A -85,B 0,C 180,E1 14411.321,E2 14411.321} C_VEL
LIN {X 0,Y 306.35,Z 702.53,A -85,B 0,C 180,E1 14417.163,E2 14417.163} C_VEL
LIN {X 0,Y 306,Z 702.53,A -85,B 0,C 180,E1 14423.205,E2 14423.205} C_VEL
LIN {X 0,Y 305.712,Z 702.53,A -85,B 0,C 180,E1 14429.544,E2 14429.544} C_VEL
LIN {X 0,Y 305.438,Z 702.53,A -85,B 0,C 180,E1 14437.77,E2 14437.77} C_VEL
LIN {X 0,Y 305.427,Z 702.53,A -85,B 0,C 180,E1 14443.72,E2 14443.72} C_VEL
LIN {X 0,Y 305.419,Z 702.53,A -85,B 0,C 180,E1 14452.181,E2 14452.181} C_VEL
LIN {X 0,Y 305.726,Z 702.53,A -85,B 0,C 180,E1 14458.432,E2 14458.432} C_VEL
LIN {X 0,Y 307.75,Z 707.795,A -85,B 0,C 180,E1 14459.248,E2 14459.248} C_VEL
LIN {X 0,Y 310.48,Z 711.077,A -85,B 0,C 180,E1 14460.142,E2 14460.142} C_VEL
LIN {X 0,Y 326.408,Z 735.304,A -85,B 0,C 180,E1 14465.167,E2 14465.167} C_VEL
LIN {X 0,Y 340.146,Z 762.391,A -85,B 0,C 180,E1 14469.777,E2 14469.777} C_VEL
LIN {X 0,Y 349.85,Z 790.355,A -85,B 0,C 180,E1 14473.993,E2 14473.993} C_VEL
LIN {X 0,Y 350.747,Z 797.747,A -85,B 0,C 180,E1 14474.915,E2 14474.915} C_VEL
LIN {X 0,Y 342.513,Z 831.738,A -85,B 0,C 180,E1 14478.082,E2 14478.082} C_VEL
LIN {X 0,Y 333.492,Z 862.565,A -85,B 0,C 180,E1 14482.198,E2 14482.198} C_VEL
LIN {X 0,Y 324.577,Z 889.541,A -85,B 0,C 180,E1 14487.336,E2 14487.336} C_VEL
LIN {X 0,Y 317.21,Z 911.345,A -85,B 0,C 180,E1 14493.253,E2 14493.253} C_VEL
LIN {X 0,Y 312.226,Z 927.45,A -85,B 0,C 180,E1 14499.627,E2 14499.627} C_VEL
LIN {X 0,Y 309.708,Z 937.211,A -85,B 0,C 180,E1 14505.545,E2 14505.545} C_VEL
LIN {X 0,Y 308.15,Z 943.002,A -85,B 0,C 180,E1 14511.593,E2 14511.593} C_VEL
LIN {X 0,Y 307.539,Z 944.837,A -85,B 0,C 180,E1 14518.041,E2 14518.041} C_VEL
LIN {X 0,Y 308.523,Z 942.753,A -85,B 0,C 180,E1 14523.809,E2 14523.809} C_VEL
LIN {X 0,Y 310.646,Z 935.743,A -85,B 0,C 180,E1 14530.518,E2 14530.518} C_VEL
LIN {X 0,Y 314.96,Z 922.614,A -85,B 0,C 180,E1 14537.517,E2 14537.517} C_VEL
LIN {X 0,Y 321.781,Z 903.882,A -85,B 0,C 180,E1 14544.005,E2 14544.005} C_VEL
LIN {X 0,Y 330.673,Z 880.168,A -85,B 0,C 180,E1 14549.596,E2 14549.596} C_VEL
LIN {X 0,Y 340.264,Z 852.508,A -85,B 0,C 180,E1 14554.189,E2 14554.189} C_VEL
LIN {X 0,Y 349.734,Z 821.085,A -85,B 0,C 180,E1 14557.878,E2 14557.878} C_VEL
LIN {X 0,Y 355.19,Z 798.74,A -85,B 0,C 180,E1 14559.84,E2 14559.84} C_VEL
LIN {X 0,Y 348.428,Z 773.445,A -85,B 0,C 180,E1 14563.997,E2 14563.997} C_VEL
LIN {X 0,Y 338.644,Z 750.336,A -85,B 0,C 180,E1 14568.621,E2 14568.621} C_VEL
LIN {X 0,Y 327.65,Z 730.881,A -85,B 0,C 180,E1 14573.909,E2 14573.909} C_VEL
LIN {X 0,Y 322.301,Z 723.535,A -85,B 0,C 180,E1 14576.86,E2 14576.86} C_VEL
LIN {X 0,Y 318.486,Z 717.374,A -85,B 0,C 180,E1 14579.513,E2 14579.513} C_VEL
LIN {X 0,Y 314.058,Z 711.819,A -85,B 0,C 180,E1 14583.637,E2 14583.637} C_VEL
LIN {X 0,Y 313.2,Z 710.2,A -85,B 0,C 180,E1 14584.858,E2 14584.858} C_VEL
LIN {X 0,Y 312.213,Z 710.115,A -85,B 0,C 180,E1 14594.834,E2 14594.834} C_VEL
LIN {X 0,Y 313.006,Z 711.267,A -85,B 0,C 180,E1 14596.228,E2 14596.228} C_VEL
LIN {X 0,Y 316.29,Z 716.784,A -85,B 0,C 180,E1 14600.073,E2 14600.073} C_VEL
LIN {X 0,Y 318.541,Z 719.083,A -85,B 0,C 180,E1 14601.831,E2 14601.831} C_VEL
LIN {X 0,Y 323.918,Z 727.013,A -85,B 0,C 180,E1 14605.288,E2 14605.288} C_VEL
LIN {X 0,Y 332.409,Z 739.339,A -85,B 0,C 180,E1 14609.4,E2 14609.4} C_VEL
LIN {X 0,Y 344.49,Z 759.403,A -85,B 0,C 180,E1 14614.151,E2 14614.151} C_VEL
LIN {X 0,Y 356.024,Z 786.095,A -85,B 0,C 180,E1 14618.613,E2 14618.613} C_VEL
LIN {X 0,Y 361.158,Z 804.78,A -85,B 0,C 180,E1 14621.098,E2 14621.098} C_VEL
LIN {X 0,Y 352.75,Z 841.677,A -85,B 0,C 180,E1 14623.567,E2 14623.567} C_VEL
LIN {X 0,Y 342.809,Z 876.414,A -85,B 0,C 180,E1 14626.962,E2 14626.962} C_VEL
LIN {X 0,Y 332.52,Z 908.333,A -85,B 0,C 180,E1 14631.391,E2 14631.391} C_VEL
LIN {X 0,Y 322.968,Z 936.7,A -85,B 0,C 180,E1 14636.872,E2 14636.872} C_VEL
LIN {X 0,Y 315.421,Z 960.76,A -85,B 0,C 180,E1 14643.351,E2 14643.351} C_VEL
LIN {X 0,Y 310.352,Z 979.87,A -85,B 0,C 180,E1 14650.698,E2 14650.698} C_VEL
LIN {X 0,Y 308.554,Z 991.102,A -85,B 0,C 180,E1 14657.152,E2 14657.152} C_VEL
LIN {X 0,Y 308.038,Z 997.355,A -85,B 0,C 180,E1 14662.965,E2 14662.965} C_VEL
LIN {X 0,Y 308.325,Z 1000.158,A -85,B 0,C 180,E1 14670,E2 14670} C_VEL
LIN {X 0,Y 308.035,Z 997.527,A -85,B 0,C 180,E1 14677.034,E2 14677.034} C_VEL
LIN {X 0,Y 308.779,Z 989.482,A -85,B 0,C 180,E1 14684.143,E2 14684.143} C_VEL
LIN {X 0,Y 311.375,Z 975.653,A -85,B 0,C 180,E1 14691.313,E2 14691.313} C_VEL
LIN {X 0,Y 317.09,Z 955.135,A -85,B 0,C 180,E1 14698.417,E2 14698.417} C_VEL
LIN {X 0,Y 324.688,Z 931.199,A -85,B 0,C 180,E1 14704.299,E2 14704.299} C_VEL
LIN {X 0,Y 334.197,Z 901.886,A -85,B 0,C 180,E1 14709.494,E2 14709.494} C_VEL
LIN {X 0,Y 337.84,Z 890.452,A -85,B 0,C 180,E1 14711.097,E2 14711.097} C_VEL
LIN {X 0,Y 338.594,Z 877.518,A -85,B 0,C 180,E1 14713.1,E2 14713.1} C_VEL
LIN {X 0,Y 339.386,Z 864.033,A -85,B 0,C 180,E1 14714.985,E2 14714.985} C_VEL
LIN {X 0,Y 348.745,Z 827.697,A -85,B 0,C 180,E1 14718.066,E2 14718.066} C_VEL
LIN {X 0,Y 353.141,Z 805.569,A -85,B 0,C 180,E1 14719.452,E2 14719.452} C_VEL
LIN {X 0,Y 341.346,Z 775.144,A -85,B 0,C 180,E1 14723.667,E2 14723.667} C_VEL
LIN {X 0,Y 325.075,Z 744.645,A -85,B 0,C 180,E1 14728.598,E2 14728.598} C_VEL
LIN {X 0,Y 308.86,Z 719.9,A -85,B 0,C 180,E1 14733.65,E2 14733.65} C_VEL
LIN {X 0,Y 301.021,Z 708.638,A -85,B 0,C 180,E1 14736.435,E2 14736.435} C_VEL
LIN {X 0,Y 298.172,Z 703.449,A -85,B 0,C 180,E1 14737.575,E2 14737.575} C_VEL
LIN {X 0,Y 298.109,Z 702.53,A -85,B 0,C 180,E1 14737.668,E2 14737.668} C_VEL
LIN {X 0,Y 298.601,Z 702.53,A -85,B 0,C 180,E1 14745.343,E2 14745.343} C_VEL
LIN {X 0,Y 299.015,Z 702.53,A -85,B 0,C 180,E1 14751.271,E2 14751.271} C_VEL
LIN {X 0,Y 299.499,Z 702.53,A -85,B 0,C 180,E1 14757.089,E2 14757.089} C_VEL
LIN {X 0,Y 299.561,Z 702.53,A -85,B 0,C 180,E1 14762.864,E2 14762.864} C_VEL
LIN {X 0,Y 298.827,Z 702.53,A -85,B 0,C 180,E1 14771.627,E2 14771.627} C_VEL
LIN {X 0,Y 298.381,Z 702.53,A -85,B 0,C 180,E1 14777.636,E2 14777.636} C_VEL
LIN {X 0,Y 297.934,Z 702.53,A -85,B 0,C 180,E1 14784.261,E2 14784.261} C_VEL
LIN {X 0,Y 297.685,Z 702.53,A -85,B 0,C 180,E1 14790.485,E2 14790.485} C_VEL
LIN {X 0,Y 297.53,Z 702.53,A -85,B 0,C 180,E1 14797.45,E2 14797.45} C_VEL
LIN {X 0,Y 297.462,Z 702.53,A -85,B 0,C 180,E1 14805.206,E2 14805.206} C_VEL
LIN {X 0,Y 297.512,Z 702.53,A -85,B 0,C 180,E1 14812.508,E2 14812.508} C_VEL
LIN {X 0,Y 297.559,Z 702.594,A -85,B 0,C 180,E1 14815.976,E2 14815.976} C_VEL
LIN {X 0,Y 299.769,Z 707.837,A -85,B 0,C 180,E1 14816.928,E2 14816.928} C_VEL
LIN {X 0,Y 302.704,Z 711.206,A -85,B 0,C 180,E1 14817.971,E2 14817.971} C_VEL
LIN {X 0,Y 318.475,Z 734.575,A -85,B 0,C 180,E1 14823.322,E2 14823.322} C_VEL
LIN {X 0,Y 332.468,Z 761.723,A -85,B 0,C 180,E1 14828.261,E2 14828.261} C_VEL
LIN {X 0,Y 342.132,Z 788.021,A -85,B 0,C 180,E1 14832.483,E2 14832.483} C_VEL
LIN {X 0,Y 344.641,Z 799.312,A -85,B 0,C 180,E1 14834.13,E2 14834.13} C_VEL
LIN {X 0,Y 336.077,Z 833.252,A -85,B 0,C 180,E1 14837.356,E2 14837.356} C_VEL
LIN {X 0,Y 326.398,Z 864.804,A -85,B 0,C 180,E1 14841.694,E2 14841.694} C_VEL
LIN {X 0,Y 317.696,Z 889.967,A -85,B 0,C 180,E1 14846.596,E2 14846.596} C_VEL
LIN {X 0,Y 310.144,Z 911.258,A -85,B 0,C 180,E1 14852.44,E2 14852.44} C_VEL
LIN {X 0,Y 304.601,Z 928.245,A -85,B 0,C 180,E1 14859.264,E2 14859.264} C_VEL
LIN {X 0,Y 301.744,Z 938.79,A -85,B 0,C 180,E1 14865.966,E2 14865.966} C_VEL
LIN {X 0,Y 300.521,Z 943.143,A -85,B 0,C 180,E1 14870.579,E2 14870.579} C_VEL
LIN {X 0,Y 299.649,Z 945.598,A -85,B 0,C 180,E1 14876.952,E2 14876.952} C_VEL
LIN {X 0,Y 300.584,Z 943.77,A -85,B 0,C 180,E1 14883.521,E2 14883.521} C_VEL
LIN {X 0,Y 302.754,Z 937.194,A -85,B 0,C 180,E1 14890.389,E2 14890.389} C_VEL
LIN {X 0,Y 307.088,Z 924.75,A -85,B 0,C 180,E1 14897.485,E2 14897.485} C_VEL
LIN {X 0,Y 313.986,Z 906.877,A -85,B 0,C 180,E1 14904.031,E2 14904.031} C_VEL
LIN {X 0,Y 323.056,Z 883.965,A -85,B 0,C 180,E1 14909.787,E2 14909.787} C_VEL
LIN {X 0,Y 333.588,Z 855.289,A -85,B 0,C 180,E1 14914.787,E2 14914.787} C_VEL
LIN {X 0,Y 343.588,Z 823.824,A -85,B 0,C 180,E1 14918.597,E2 14918.597} C_VEL
LIN {X 0,Y 349.363,Z 802.065,A -85,B 0,C 180,E1 14920.551,E2 14920.551} C_VEL
LIN {X 0,Y 343.016,Z 776.769,A -85,B 0,C 180,E1 14924.93,E2 14924.93} C_VEL
LIN {X 0,Y 333.773,Z 753.991,A -85,B 0,C 180,E1 14929.769,E2 14929.769} C_VEL
LIN {X 0,Y 324.482,Z 737.297,A -85,B 0,C 180,E1 14934.686,E2 14934.686} C_VEL
LIN {X 0,Y 319.853,Z 730.299,A -85,B 0,C 180,E1 14937.54,E2 14937.54} C_VEL
LIN {X 0,Y 316.636,Z 724.78,A -85,B 0,C 180,E1 14940.022,E2 14940.022} C_VEL
LIN {X 0,Y 312.558,Z 719,A -85,B 0,C 180,E1 14944.174,E2 14944.174} C_VEL
LIN {X 0,Y 310.297,Z 717.439,A -85,B 0,C 180,E1 14948.41,E2 14948.41} C_VEL
LIN {X 0,Y 311.675,Z 718.755,A -85,B 0,C 180,E1 14955.817,E2 14955.817} C_VEL
LIN {X 0,Y 314.883,Z 724.434,A -85,B 0,C 180,E1 14959.801,E2 14959.801} C_VEL
LIN {X 0,Y 317.036,Z 727.028,A -85,B 0,C 180,E1 14961.573,E2 14961.573} C_VEL
LIN {X 0,Y 322.354,Z 735.021,A -85,B 0,C 180,E1 14965.096,E2 14965.096} C_VEL
LIN {X 0,Y 330.261,Z 747.065,A -85,B 0,C 180,E1 14969.104,E2 14969.104} C_VEL
LIN {X 0,Y 340.774,Z 765.667,A -85,B 0,C 180,E1 14973.625,E2 14973.625} C_VEL
LIN {X 0,Y 351.287,Z 791.758,A -85,B 0,C 180,E1 14978.124,E2 14978.124} C_VEL
LIN {X 0,Y 355.399,Z 806.804,A -85,B 0,C 180,E1 14980.266,E2 14980.266} C_VEL
LIN {X 0,Y 346.758,Z 842.849,A -85,B 0,C 180,E1 14982.746,E2 14982.746} C_VEL
LIN {X 0,Y 336.228,Z 877.828,A -85,B 0,C 180,E1 14986.26,E2 14986.26} C_VEL
LIN {X 0,Y 325.46,Z 909.62,A -85,B 0,C 180,E1 14990.821,E2 14990.821} C_VEL
LIN {X 0,Y 315.67,Z 937.212,A -85,B 0,C 180,E1 14996.334,E2 14996.334} C_VEL
LIN {X 0,Y 307.607,Z 961.637,A -85,B 0,C 180,E1 15003.185,E2 15003.185} C_VEL
LIN {X 0,Y 302.692,Z 979.118,A -85,B 0,C 180,E1 15010.173,E2 15010.173} C_VEL
LIN {X 0,Y 300.68,Z 990.579,A -85,B 0,C 180,E1 15016.947,E2 15016.947} C_VEL
LIN {X 0,Y 300.155,Z 996.643,A -85,B 0,C 180,E1 15022.779,E2 15022.779} C_VEL
LIN {X 0,Y 300.473,Z 999.449,A -85,B 0,C 180,E1 15030,E2 15030} C_VEL
LIN {X 0,Y 300.15,Z 996.804,A -85,B 0,C 180,E1 15037.22,E2 15037.22} C_VEL
LIN {X 0,Y 300.96,Z 988.726,A -85,B 0,C 180,E1 15044.519,E2 15044.519} C_VEL
LIN {X 0,Y 303.755,Z 974.838,A -85,B 0,C 180,E1 15051.875,E2 15051.875} C_VEL
LIN {X 0,Y 309.836,Z 954.222,A -85,B 0,C 180,E1 15059.146,E2 15059.146} C_VEL
LIN {X 0,Y 318.228,Z 929.213,A -85,B 0,C 180,E1 15065.338,E2 15065.338} C_VEL
LIN {X 0,Y 327.874,Z 900.708,A -85,B 0,C 180,E1 15070.41,E2 15070.41} C_VEL
LIN {X 0,Y 338.071,Z 868.534,A -85,B 0,C 180,E1 15074.502,E2 15074.502} C_VEL
LIN {X 0,Y 339.386,Z 864.033,A -85,B 0,C 180,E1 15074.985,E2 15074.985} C_VEL
LIN {X 0,Y 340.201,Z 850.001,A -85,B 0,C 180,E1 15076.758,E2 15076.758} C_VEL
LIN {X 0,Y 340.949,Z 835.429,A -85,B 0,C 180,E1 15078.382,E2 15078.382} C_VEL
LIN {X 0,Y 346.793,Z 808.029,A -85,B 0,C 180,E1 15080.236,E2 15080.236} C_VEL
LIN {X 0,Y 335.239,Z 777.603,A -85,B 0,C 180,E1 15084.664,E2 15084.664} C_VEL
LIN {X 0,Y 320.175,Z 748.942,A -85,B 0,C 180,E1 15089.541,E2 15089.541} C_VEL
LIN {X 0,Y 303.076,Z 722.261,A -85,B 0,C 180,E1 15095.191,E2 15095.191} C_VEL
LIN {X 0,Y 293.656,Z 709.005,A -85,B 0,C 180,E1 15098.799,E2 15098.799} C_VEL
LIN {X 0,Y 290.461,Z 704.253,A -85,B 0,C 180,E1 15100.159,E2 15100.159} C_VEL
LIN {X 0,Y 290.281,Z 702.53,A -85,B 0,C 180,E1 15100.364,E2 15100.364} C_VEL
LIN {X 0,Y 290.862,Z 702.53,A -85,B 0,C 180,E1 15108.001,E2 15108.001} C_VEL
LIN {X 0,Y 291.575,Z 702.53,A -85,B 0,C 180,E1 15117.01,E2 15117.01} C_VEL
LIN {X 0,Y 291.636,Z 702.53,A -85,B 0,C 180,E1 15122.941,E2 15122.941} C_VEL
LIN {X 0,Y 290.867,Z 702.53,A -85,B 0,C 180,E1 15131.95,E2 15131.95} C_VEL
LIN {X 0,Y 290.286,Z 702.53,A -85,B 0,C 180,E1 15140.657,E2 15140.657} C_VEL
LIN {X 0,Y 289.831,Z 702.53,A -85,B 0,C 180,E1 15147.909,E2 15147.909} C_VEL
LIN {X 0,Y 289.616,Z 702.53,A -85,B 0,C 180,E1 15154.931,E2 15154.931} C_VEL
LIN {X 0,Y 289.432,Z 702.53,A -85,B 0,C 180,E1 15163.121,E2 15163.121} C_VEL
LIN {X 0,Y 289.521,Z 702.53,A -85,B 0,C 180,E1 15171.372,E2 15171.372} C_VEL
LIN {X 0,Y 289.613,Z 703.14,A -85,B 0,C 180,E1 15173.321,E2 15173.321} C_VEL
LIN {X 0,Y 292.139,Z 708.327,A -85,B 0,C 180,E1 15174.49,E2 15174.49} C_VEL
LIN {X 0,Y 294.76,Z 711.205,A -85,B 0,C 180,E1 15175.512,E2 15175.512} C_VEL
LIN {X 0,Y 311.324,Z 735.372,A -85,B 0,C 180,E1 15181.612,E2 15181.612} C_VEL
LIN {X 0,Y 325.328,Z 761.97,A -85,B 0,C 180,E1 15186.833,E2 15186.833} C_VEL
LIN {X 0,Y 335.388,Z 788.883,A -85,B 0,C 180,E1 15191.4,E2 15191.4} C_VEL
LIN {X 0,Y 338.536,Z 801.049,A -85,B 0,C 180,E1 15193.325,E2 15193.325} C_VEL
LIN {X 0,Y 329.679,Z 834.765,A -85,B 0,C 180,E1 15196.602,E2 15196.602} C_VEL
LIN {X 0,Y 319.669,Z 866.018,A -85,B 0,C 180,E1 15201.001,E2 15201.001} C_VEL
LIN {X 0,Y 310.242,Z 892.16,A -85,B 0,C 180,E1 15206.253,E2 15206.253} C_VEL
LIN {X 0,Y 302.301,Z 913.597,A -85,B 0,C 180,E1 15212.406,E2 15212.406} C_VEL
LIN {X 0,Y 296.551,Z 930.197,A -85,B 0,C 180,E1 15219.52,E2 15219.52} C_VEL
LIN {X 0,Y 293.747,Z 940.228,A -85,B 0,C 180,E1 15226.413,E2 15226.413} C_VEL
LIN {X 0,Y 292.304,Z 944.659,A -85,B 0,C 180,E1 15231.78,E2 15231.78} C_VEL
LIN {X 0,Y 291.81,Z 946.242,A -85,B 0,C 180,E1 15238.539,E2 15238.539} C_VEL
LIN {X 0,Y 293.479,Z 942.739,A -85,B 0,C 180,E1 15246.232,E2 15246.232} C_VEL
LIN {X 0,Y 296.21,Z 934.762,A -85,B 0,C 180,E1 15253.04,E2 15253.04} C_VEL
LIN {X 0,Y 301.436,Z 921.189,A -85,B 0,C 180,E1 15259.967,E2 15259.967} C_VEL
LIN {X 0,Y 309.552,Z 901.666,A -85,B 0,C 180,E1 15266.515,E2 15266.515} C_VEL
LIN {X 0,Y 319.247,Z 878.146,A -85,B 0,C 180,E1 15271.965,E2 15271.965} C_VEL
LIN {X 0,Y 330.25,Z 848.929,A -85,B 0,C 180,E1 15276.704,E2 15276.704} C_VEL
LIN {X 0,Y 340.371,Z 816.929,A -85,B 0,C 180,E1 15280.299,E2 15280.299} C_VEL
LIN {X 0,Y 343.544,Z 805.413,A -85,B 0,C 180,E1 15281.293,E2 15281.293} C_VEL
LIN {X 0,Y 337.779,Z 780.514,A -85,B 0,C 180,E1 15285.801,E2 15285.801} C_VEL
LIN {X 0,Y 329.37,Z 758.766,A -85,B 0,C 180,E1 15290.713,E2 15290.713} C_VEL
LIN {X 0,Y 321.523,Z 743.806,A -85,B 0,C 180,E1 15295.365,E2 15295.365} C_VEL
LIN {X 0,Y 317.339,Z 736.976,A -85,B 0,C 180,E1 15298.271,E2 15298.271} C_VEL
LIN {X 0,Y 314.654,Z 732.146,A -85,B 0,C 180,E1 15300.537,E2 15300.537} C_VEL
LIN {X 0,Y 310.521,Z 725.675,A -85,B 0,C 180,E1 15305.599,E2 15305.599} C_VEL
LIN {X 0,Y 310.308,Z 725.952,A -85,B 0,C 180,E1 15315.262,E2 15315.262} C_VEL
LIN {X 0,Y 313.283,Z 731.919,A -85,B 0,C 180,E1 15319.358,E2 15319.358} C_VEL
LIN {X 0,Y 315.398,Z 734.572,A -85,B 0,C 180,E1 15321.213,E2 15321.213} C_VEL
LIN {X 0,Y 320.662,Z 742.902,A -85,B 0,C 180,E1 15324.902,E2 15324.902} C_VEL
LIN {X 0,Y 329.867,Z 758.067,A -85,B 0,C 180,E1 15329.803,E2 15329.803} C_VEL
LIN {X 0,Y 339.181,Z 776.908,A -85,B 0,C 180,E1 15334.092,E2 15334.092} C_VEL
LIN {X 0,Y 347.943,Z 802.393,A -85,B 0,C 180,E1 15338.404,E2 15338.404} C_VEL
LIN {X 0,Y 349.261,Z 810.988,A -85,B 0,C 180,E1 15339.517,E2 15339.517} C_VEL
LIN {X 0,Y 339.397,Z 849.181,A -85,B 0,C 180,E1 15342.338,E2 15342.338} C_VEL
LIN {X 0,Y 328.158,Z 883.88,A -85,B 0,C 180,E1 15346.119,E2 15346.119} C_VEL
LIN {X 0,Y 317.04,Z 914.66,A -85,B 0,C 180,E1 15350.9,E2 15350.9} C_VEL
LIN {X 0,Y 307.07,Z 941.319,A -85,B 0,C 180,E1 15356.681,E2 15356.681} C_VEL
LIN {X 0,Y 299.296,Z 963.561,A -85,B 0,C 180,E1 15363.418,E2 15363.418} C_VEL
LIN {X 0,Y 294.537,Z 980.373,A -85,B 0,C 180,E1 15370.67,E2 15370.67} C_VEL
LIN {X 0,Y 292.847,Z 989.872,A -85,B 0,C 180,E1 15376.592,E2 15376.592} C_VEL
LIN {X 0,Y 292.289,Z 995.937,A -85,B 0,C 180,E1 15382.584,E2 15382.584} C_VEL
LIN {X 0,Y 292.62,Z 998.74,A -85,B 0,C 180,E1 15390,E2 15390} C_VEL
LIN {X 0,Y 292.282,Z 996.081,A -85,B 0,C 180,E1 15397.416,E2 15397.416} C_VEL
LIN {X 0,Y 293.175,Z 987.962,A -85,B 0,C 180,E1 15404.913,E2 15404.913} C_VEL
LIN {X 0,Y 296.14,Z 974.09,A -85,B 0,C 180,E1 15412.431,E2 15412.431} C_VEL
LIN {X 0,Y 302.162,Z 954.754,A -85,B 0,C 180,E1 15419.482,E2 15419.482} C_VEL
LIN {X 0,Y 311.008,Z 929.594,A -85,B 0,C 180,E1 15425.917,E2 15425.917} C_VEL
LIN {X 0,Y 321.133,Z 901.007,A -85,B 0,C 180,E1 15431.137,E2 15431.137} C_VEL
LIN {X 0,Y 331.751,Z 868.721,A -85,B 0,C 180,E1 15435.318,E2 15435.318} C_VEL
LIN {X 0,Y 340.949,Z 835.429,A -85,B 0,C 180,E1 15438.382,E2 15438.382} C_VEL
LIN {X 0,Y 342.335,Z 823.859,A -85,B 0,C 180,E1 15439.437,E2 15439.437} C_VEL
LIN {X 0,Y 339.184,Z 806.218,A -85,B 0,C 180,E1 15441.66,E2 15441.66} C_VEL
LIN {X 0,Y 327.203,Z 775.86,A -85,B 0,C 180,E1 15446.381,E2 15446.381} C_VEL
LIN {X 0,Y 311.476,Z 746.483,A -85,B 0,C 180,E1 15451.786,E2 15451.786} C_VEL
LIN {X 0,Y 295.196,Z 722.083,A -85,B 0,C 180,E1 15457.634,E2 15457.634} C_VEL
LIN {X 0,Y 285.848,Z 708.975,A -85,B 0,C 180,E1 15461.611,E2 15461.611} C_VEL
LIN {X 0,Y 282.695,Z 704.216,A -85,B 0,C 180,E1 15463.129,E2 15463.129} C_VEL
LIN {X 0,Y 282.531,Z 702.53,A -85,B 0,C 180,E1 15463.523,E2 15463.523} C_VEL
LIN {X 0,Y 283.128,Z 702.53,A -85,B 0,C 180,E1 15470.777,E2 15470.777} C_VEL
LIN {X 0,Y 283.65,Z 702.53,A -85,B 0,C 180,E1 15476.927,E2 15476.927} C_VEL
LIN {X 0,Y 283.73,Z 702.53,A -85,B 0,C 180,E1 15483.024,E2 15483.024} C_VEL
LIN {X 0,Y 282.898,Z 702.53,A -85,B 0,C 180,E1 15492.292,E2 15492.292} C_VEL
LIN {X 0,Y 282.418,Z 702.53,A -85,B 0,C 180,E1 15498.668,E2 15498.668} C_VEL
LIN {X 0,Y 281.982,Z 702.53,A -85,B 0,C 180,E1 15505.315,E2 15505.315} C_VEL
LIN {X 0,Y 281.725,Z 702.53,A -85,B 0,C 180,E1 15512.349,E2 15512.349} C_VEL
LIN {X 0,Y 281.458,Z 702.53,A -85,B 0,C 180,E1 15520,E2 15520} C_VEL
LIN {X 0,Y 281.435,Z 702.53,A -85,B 0,C 180,E1 15528.595,E2 15528.595} C_VEL
LIN {X 0,Y 281.452,Z 702.53,A -85,B 0,C 180,E1 15530.161,E2 15530.161} C_VEL
LIN {X 0,Y 283.318,Z 707.427,A -85,B 0,C 180,E1 15531.217,E2 15531.217} C_VEL
LIN {X 0,Y 286.934,Z 711.292,A -85,B 0,C 180,E1 15532.81,E2 15532.81} C_VEL
LIN {X 0,Y 300.552,Z 730.565,A -85,B 0,C 180,E1 15538.346,E2 15538.346} C_VEL
LIN {X 0,Y 314.103,Z 753.697,A -85,B 0,C 180,E1 15543.621,E2 15543.621} C_VEL
LIN {X 0,Y 325.506,Z 780.162,A -85,B 0,C 180,E1 15548.607,E2 15548.607} C_VEL
LIN {X 0,Y 332.103,Z 803.202,A -85,B 0,C 180,E1 15552.481,E2 15552.481} C_VEL
LIN {X 0,Y 322.933,Z 837.544,A -85,B 0,C 180,E1 15555.972,E2 15555.972} C_VEL
LIN {X 0,Y 312.894,Z 867.441,A -85,B 0,C 180,E1 15560.312,E2 15560.312} C_VEL
LIN {X 0,Y 303.274,Z 892.97,A -85,B 0,C 180,E1 15565.553,E2 15565.553} C_VEL
LIN {X 0,Y 294.948,Z 914.42,A -85,B 0,C 180,E1 15571.849,E2 15571.849} C_VEL
LIN {X 0,Y 289.005,Z 930.754,A -85,B 0,C 180,E1 15579.013,E2 15579.013} C_VEL
LIN {X 0,Y 286.232,Z 940.013,A -85,B 0,C 180,E1 15585.284,E2 15585.284} C_VEL
LIN {X 0,Y 284.422,Z 945.437,A -85,B 0,C 180,E1 15591.802,E2 15591.802} C_VEL
LIN {X 0,Y 283.959,Z 946.957,A -85,B 0,C 180,E1 15598.574,E2 15598.574} C_VEL
LIN {X 0,Y 285.408,Z 944.166,A -85,B 0,C 180,E1 15605.564,E2 15605.564} C_VEL
LIN {X 0,Y 288.265,Z 936.409,A -85,B 0,C 180,E1 15612.886,E2 15612.886} C_VEL
LIN {X 0,Y 293.939,Z 922.61,A -85,B 0,C 180,E1 15620.361,E2 15620.361} C_VEL
LIN {X 0,Y 302.496,Z 903.205,A -85,B 0,C 180,E1 15627.105,E2 15627.105} C_VEL
LIN {X 0,Y 312.749,Z 879.538,A -85,B 0,C 180,E1 15632.741,E2 15632.741} C_VEL
LIN {X 0,Y 323.683,Z 851.936,A -85,B 0,C 180,E1 15637.356,E2 15637.356} C_VEL
LIN {X 0,Y 334.775,Z 818.855,A -85,B 0,C 180,E1 15641.191,E2 15641.191} C_VEL
LIN {X 0,Y 337.798,Z 808.301,A -85,B 0,C 180,E1 15642.14,E2 15642.14} C_VEL
LIN {X 0,Y 332.767,Z 784.881,A -85,B 0,C 180,E1 15646.586,E2 15646.586} C_VEL
LIN {X 0,Y 325.229,Z 763.955,A -85,B 0,C 180,E1 15651.553,E2 15651.553} C_VEL
LIN {X 0,Y 318.148,Z 749.628,A -85,B 0,C 180,E1 15656.296,E2 15656.296} C_VEL
LIN {X 0,Y 312.806,Z 739.63,A -85,B 0,C 180,E1 15660.886,E2 15660.886} C_VEL
LIN {X 0,Y 309.263,Z 733.473,A -85,B 0,C 180,E1 15665.622,E2 15665.622} C_VEL
LIN {X 0,Y 309.003,Z 733.947,A -85,B 0,C 180,E1 15675.056,E2 15675.056} C_VEL
LIN {X 0,Y 312.649,Z 740.258,A -85,B 0,C 180,E1 15679.902,E2 15679.902} C_VEL
LIN {X 0,Y 318.905,Z 750.917,A -85,B 0,C 180,E1 15684.816,E2 15684.816} C_VEL
LIN {X 0,Y 327.202,Z 765.784,A -85,B 0,C 180,E1 15689.581,E2 15689.581} C_VEL
LIN {X 0,Y 335.937,Z 785.028,A -85,B 0,C 180,E1 15693.981,E2 15693.981} C_VEL
LIN {X 0,Y 343.571,Z 810.695,A -85,B 0,C 180,E1 15698.36,E2 15698.36} C_VEL
LIN {X 0,Y 342.425,Z 818.027,A -85,B 0,C 180,E1 15698.948,E2 15698.948} C_VEL
LIN {X 0,Y 332.35,Z 854.065,A -85,B 0,C 180,E1 15701.831,E2 15701.831} C_VEL
LIN {X 0,Y 320.994,Z 887.065,A -85,B 0,C 180,E1 15705.63,E2 15705.63} C_VEL
LIN {X 0,Y 309.277,Z 917.642,A -85,B 0,C 180,E1 15710.632,E2 15710.632} C_VEL
LIN {X 0,Y 298.95,Z 943.992,A -85,B 0,C 180,E1 15716.705,E2 15716.705} C_VEL
LIN {X 0,Y 290.914,Z 965.947,A -85,B 0,C 180,E1 15723.838,E2 15723.838} C_VEL
LIN {X 0,Y 286.222,Z 982.424,A -85,B 0,C 180,E1 15731.658,E2 15731.658} C_VEL
LIN {X 0,Y 284.711,Z 991.866,A -85,B 0,C 180,E1 15738.561,E2 15738.561} C_VEL
LIN {X 0,Y 284.37,Z 996.206,A -85,B 0,C 180,E1 15743.907,E2 15743.907} C_VEL
LIN {X 0,Y 284.749,Z 998.028,A -85,B 0,C 180,E1 15750,E2 15750} C_VEL
LIN {X 0,Y 284.408,Z 995.35,A -85,B 0,C 180,E1 15757.622,E2 15757.622} C_VEL
LIN {X 0,Y 285.369,Z 987.19,A -85,B 0,C 180,E1 15765.331,E2 15765.331} C_VEL
LIN {X 0,Y 288.526,Z 973.463,A -85,B 0,C 180,E1 15772.955,E2 15772.955} C_VEL
LIN {X 0,Y 294.979,Z 953.817,A -85,B 0,C 180,E1 15780.269,E2 15780.269} C_VEL
LIN {X 0,Y 303.91,Z 929.744,A -85,B 0,C 180,E1 15786.572,E2 15786.572} C_VEL
LIN {X 0,Y 314.568,Z 900.848,A -85,B 0,C 180,E1 15791.957,E2 15791.957} C_VEL
LIN {X 0,Y 325.462,Z 869.016,A -85,B 0,C 180,E1 15796.154,E2 15796.154} C_VEL
LIN {X 0,Y 335.28,Z 834.808,A -85,B 0,C 180,E1 15799.334,E2 15799.334} C_VEL
LIN {X 0,Y 340.626,Z 810.939,A -85,B 0,C 180,E1 15800.979,E2 15800.979} C_VEL
LIN {X 0,Y 339.184,Z 806.218,A -85,B 0,C 180,E1 15801.66,E2 15801.66} C_VEL
LIN {X 0,Y 334.368,Z 798.3,A -85,B 0,C 180,E1 15803.238,E2 15803.238} C_VEL
LIN {X 0,Y 324.797,Z 786.58,A -85,B 0,C 180,E1 15806.049,E2 15806.049} C_VEL
LIN {X 0,Y 310.552,Z 757.559,A -85,B 0,C 180,E1 15811.391,E2 15811.391} C_VEL
LIN {X 0,Y 295.741,Z 733.843,A -85,B 0,C 180,E1 15816.893,E2 15816.893} C_VEL
LIN {X 0,Y 283.425,Z 716.101,A -85,B 0,C 180,E1 15822.152,E2 15822.152} C_VEL
LIN {X 0,Y 279.692,Z 710.221,A -85,B 0,C 180,E1 15824.012,E2 15824.012} C_VEL
LIN {X 0,Y 275.264,Z 705.242,A -85,B 0,C 180,E1 15826.302,E2 15826.302} C_VEL
LIN {X 0,Y 274.854,Z 702.53,A -85,B 0,C 180,E1 15826.888,E2 15826.888} C_VEL
LIN {X 0,Y 275.417,Z 702.53,A -85,B 0,C 180,E1 15833.685,E2 15833.685} C_VEL
LIN {X 0,Y 275.968,Z 702.53,A -85,B 0,C 180,E1 15839.975,E2 15839.975} C_VEL
LIN {X 0,Y 275.438,Z 702.53,A -85,B 0,C 180,E1 15846.264,E2 15846.264} C_VEL
LIN {X 0,Y 274.935,Z 702.53,A -85,B 0,C 180,E1 15852.653,E2 15852.653} C_VEL
LIN {X 0,Y 274.255,Z 702.53,A -85,B 0,C 180,E1 15860.71,E2 15860.71} C_VEL
LIN {X 0,Y 273.844,Z 702.53,A -85,B 0,C 180,E1 15869.695,E2 15869.695} C_VEL
LIN {X 0,Y 273.543,Z 702.53,A -85,B 0,C 180,E1 15877.318,E2 15877.318} C_VEL
LIN {X 0,Y 273.529,Z 702.53,A -85,B 0,C 180,E1 15885.773,E2 15885.773} C_VEL
LIN {X 0,Y 273.484,Z 702.964,A -85,B 0,C 180,E1 15886.659,E2 15886.659} C_VEL
LIN {X 0,Y 275.547,Z 707.822,A -85,B 0,C 180,E1 15887.966,E2 15887.966} C_VEL
LIN {X 0,Y 278.997,Z 711.229,A -85,B 0,C 180,E1 15889.693,E2 15889.693} C_VEL
LIN {X 0,Y 289.62,Z 726.047,A -85,B 0,C 180,E1 15894.628,E2 15894.628} C_VEL
LIN {X 0,Y 303.267,Z 747.065,A -85,B 0,C 180,E1 15900.32,E2 15900.32} C_VEL
LIN {X 0,Y 315.458,Z 772.453,A -85,B 0,C 180,E1 15905.677,E2 15905.677} C_VEL
LIN {X 0,Y 323.952,Z 797.62,A -85,B 0,C 180,E1 15910.28,E2 15910.28} C_VEL
LIN {X 0,Y 325.536,Z 808.469,A -85,B 0,C 180,E1 15911.985,E2 15911.985} C_VEL
LIN {X 0,Y 315.789,Z 841.404,A -85,B 0,C 180,E1 15915.471,E2 15915.471} C_VEL
LIN {X 0,Y 305.199,Z 871.343,A -85,B 0,C 180,E1 15920.033,E2 15920.033} C_VEL
LIN {X 0,Y 294.976,Z 897.313,A -85,B 0,C 180,E1 15925.723,E2 15925.723} C_VEL
LIN {X 0,Y 286.725,Z 917.513,A -85,B 0,C 180,E1 15932.14,E2 15932.14} C_VEL
LIN {X 0,Y 280.951,Z 932.668,A -85,B 0,C 180,E1 15939.273,E2 15939.273} C_VEL
LIN {X 0,Y 277.851,Z 942.784,A -85,B 0,C 180,E1 15947.063,E2 15947.063} C_VEL
LIN {X 0,Y 276.412,Z 946.55,A -85,B 0,C 180,E1 15952.468,E2 15952.468} C_VEL
LIN {X 0,Y 276.151,Z 947.628,A -85,B 0,C 180,E1 15959.46,E2 15959.46} C_VEL
LIN {X 0,Y 277.891,Z 944.326,A -85,B 0,C 180,E1 15966.68,E2 15966.68} C_VEL
LIN {X 0,Y 281.185,Z 936.002,A -85,B 0,C 180,E1 15974.241,E2 15974.241} C_VEL
LIN {X 0,Y 287.697,Z 921.368,A -85,B 0,C 180,E1 15981.886,E2 15981.886} C_VEL
LIN {X 0,Y 296.433,Z 902.705,A -85,B 0,C 180,E1 15988.31,E2 15988.31} C_VEL
LIN {X 0,Y 307.111,Z 879.237,A -85,B 0,C 180,E1 15993.902,E2 15993.902} C_VEL
LIN {X 0,Y 318.945,Z 850.536,A -85,B 0,C 180,E1 15998.663,E2 15998.663} C_VEL
LIN {X 0,Y 330.089,Z 818.15,A -85,B 0,C 180,E1 16002.354,E2 16002.354} C_VEL
LIN {X 0,Y 331.986,Z 810.314,A -85,B 0,C 180,E1 16003.183,E2 16003.183} C_VEL
LIN {X 0,Y 327.418,Z 787.76,A -85,B 0,C 180,E1 16007.717,E2 16007.717} C_VEL
LIN {X 0,Y 320.513,Z 767.539,A -85,B 0,C 180,E1 16012.886,E2 16012.886} C_VEL
LIN {X 0,Y 313.631,Z 752.804,A -85,B 0,C 180,E1 16018.299,E2 16018.299} C_VEL
LIN {X 0,Y 310.589,Z 746.984,A -85,B 0,C 180,E1 16021.414,E2 16021.414} C_VEL
LIN {X 0,Y 307.87,Z 741.233,A -85,B 0,C 180,E1 16025.647,E2 16025.647} C_VEL
LIN {X 0,Y 307.639,Z 741.766,A -85,B 0,C 180,E1 16034.852,E2 16034.852} C_VEL
LIN {X 0,Y 311.936,Z 750.026,A -85,B 0,C 180,E1 16040.733,E2 16040.733} C_VEL
LIN {X 0,Y 317.947,Z 760.564,A -85,B 0,C 180,E1 16045.394,E2 16045.394} C_VEL
LIN {X 0,Y 327.299,Z 779.499,A -85,B 0,C 180,E1 16050.971,E2 16050.971} C_VEL
LIN {X 0,Y 335.094,Z 802.089,A -85,B 0,C 180,E1 16055.54,E2 16055.54} C_VEL
LIN {X 0,Y 338.044,Z 815.64,A -85,B 0,C 180,E1 16057.759,E2 16057.759} C_VEL
LIN {X 0,Y 327.748,Z 851.303,A -85,B 0,C 180,E1 16060.547,E2 16060.547} C_VEL
LIN {X 0,Y 315.648,Z 885.353,A -85,B 0,C 180,E1 16064.428,E2 16064.428} C_VEL
LIN {X 0,Y 303.587,Z 915.467,A -85,B 0,C 180,E1 16069.337,E2 16069.337} C_VEL
LIN {X 0,Y 292.636,Z 941.965,A -85,B 0,C 180,E1 16075.442,E2 16075.442} C_VEL
LIN {X 0,Y 283.958,Z 964.247,A -85,B 0,C 180,E1 16082.719,E2 16082.719} C_VEL
LIN {X 0,Y 278.545,Z 981.561,A -85,B 0,C 180,E1 16091.031,E2 16091.031} C_VEL
LIN {X 0,Y 276.768,Z 991.96,A -85,B 0,C 180,E1 16098.998,E2 16098.998} C_VEL
LIN {X 0,Y 276.539,Z 996.853,A -85,B 0,C 180,E1 16106.872,E2 16106.872} C_VEL
LIN {X 0,Y 276.895,Z 997.317,A -85,B 0,C 180,E1 16110,E2 16110} C_VEL
LIN {X 0,Y 276.527,Z 994.616,A -85,B 0,C 180,E1 16117.841,E2 16117.841} C_VEL
LIN {X 0,Y 277.572,Z 986.413,A -85,B 0,C 180,E1 16125.773,E2 16125.773} C_VEL
LIN {X 0,Y 281.117,Z 972.29,A -85,B 0,C 180,E1 16133.752,E2 16133.752} C_VEL
LIN {X 0,Y 287.938,Z 952.721,A -85,B 0,C 180,E1 16141.142,E2 16141.142} C_VEL
LIN {X 0,Y 297.307,Z 928.64,A -85,B 0,C 180,E1 16147.522,E2 16147.522} C_VEL
LIN {X 0,Y 308.38,Z 899.821,A -85,B 0,C 180,E1 16152.949,E2 16152.949} C_VEL
LIN {X 0,Y 319.573,Z 868.155,A -85,B 0,C 180,E1 16157.15,E2 16157.15} C_VEL
LIN {X 0,Y 329.845,Z 833.359,A -85,B 0,C 180,E1 16160.38,E2 16160.38} C_VEL
LIN {X 0,Y 334.469,Z 813.704,A -85,B 0,C 180,E1 16161.764,E2 16161.764} C_VEL
LIN {X 0,Y 324.797,Z 786.58,A -85,B 0,C 180,E1 16166.049,E2 16166.049} C_VEL
LIN {X 0,Y 319.362,Z 779.52,A -85,B 0,C 180,E1 16167.769,E2 16167.769} C_VEL
LIN {X 0,Y 310.298,Z 770.546,A -85,B 0,C 180,E1 16170.555,E2 16170.555} C_VEL
LIN {X 0,Y 309.539,Z 769.18,A -85,B 0,C 180,E1 16170.843,E2 16170.843} C_VEL
LIN {X 0,Y 294.319,Z 742.508,A -85,B 0,C 180,E1 16176.877,E2 16176.877} C_VEL
LIN {X 0,Y 280.424,Z 722.623,A -85,B 0,C 180,E1 16182.964,E2 16182.964} C_VEL
LIN {X 0,Y 275.666,Z 716.037,A -85,B 0,C 180,E1 16185.413,E2 16185.413} C_VEL
LIN {X 0,Y 271.277,Z 709.526,A -85,B 0,C 180,E1 16187.936,E2 16187.936} C_VEL
LIN {X 0,Y 267.712,Z 705.321,A -85,B 0,C 180,E1 16190.138,E2 16190.138} C_VEL
LIN {X 0,Y 267.317,Z 702.53,A -85,B 0,C 180,E1 16190.8,E2 16190.8} C_VEL
LIN {X 0,Y 268.061,Z 702.53,A -85,B 0,C 180,E1 16199.974,E2 16199.974} C_VEL
LIN {X 0,Y 267.498,Z 702.53,A -85,B 0,C 180,E1 16206.451,E2 16206.451} C_VEL
LIN {X 0,Y 266.957,Z 702.53,A -85,B 0,C 180,E1 16213.038,E2 16213.038} C_VEL
LIN {X 0,Y 266.421,Z 702.53,A -85,B 0,C 180,E1 16219.835,E2 16219.835} C_VEL
LIN {X 0,Y 265.97,Z 702.53,A -85,B 0,C 180,E1 16226.958,E2 16226.958} C_VEL
LIN {X 0,Y 265.669,Z 702.53,A -85,B 0,C 180,E1 16234.57,E2 16234.57} C_VEL
LIN {X 0,Y 265.6,Z 703.041,A -85,B 0,C 180,E1 16242.496,E2 16242.496} C_VEL
LIN {X 0,Y 267.763,Z 707.922,A -85,B 0,C 180,E1 16244.111,E2 16244.111} C_VEL
LIN {X 0,Y 271.025,Z 710.872,A -85,B 0,C 180,E1 16246.035,E2 16246.035} C_VEL
LIN {X 0,Y 275.228,Z 716.647,A -85,B 0,C 180,E1 16248.417,E2 16248.417} C_VEL
LIN {X 0,Y 286.293,Z 732.046,A -85,B 0,C 180,E1 16253.849,E2 16253.849} C_VEL
LIN {X 0,Y 299.609,Z 753.87,A -85,B 0,C 180,E1 16259.877,E2 16259.877} C_VEL
LIN {X 0,Y 310.445,Z 777.543,A -85,B 0,C 180,E1 16265.07,E2 16265.07} C_VEL
LIN {X 0,Y 318.426,Z 803.105,A -85,B 0,C 180,E1 16269.923,E2 16269.923} C_VEL
LIN {X 0,Y 319.504,Z 810.423,A -85,B 0,C 180,E1 16271.135,E2 16271.135} C_VEL
LIN {X 0,Y 309.546,Z 842.765,A -85,B 0,C 180,E1 16274.629,E2 16274.629} C_VEL
LIN {X 0,Y 298.394,Z 873.007,A -85,B 0,C 180,E1 16279.342,E2 16279.342} C_VEL
LIN {X 0,Y 288.057,Z 898.059,A -85,B 0,C 180,E1 16284.97,E2 16284.97} C_VEL
LIN {X 0,Y 279.57,Z 917.911,A -85,B 0,C 180,E1 16291.39,E2 16291.39} C_VEL
LIN {X 0,Y 273.536,Z 932.925,A -85,B 0,C 180,E1 16298.56,E2 16298.56} C_VEL
LIN {X 0,Y 270.206,Z 942.89,A -85,B 0,C 180,E1 16306.215,E2 16306.215} C_VEL
LIN {X 0,Y 268.401,Z 947.536,A -85,B 0,C 180,E1 16313.177,E2 16313.177} C_VEL
LIN {X 0,Y 268.366,Z 948.188,A -85,B 0,C 180,E1 16320.403,E2 16320.403} C_VEL
LIN {X 0,Y 270.423,Z 944.408,A -85,B 0,C 180,E1 16327.867,E2 16327.867} C_VEL
LIN {X 0,Y 274.27,Z 935.42,A -85,B 0,C 180,E1 16335.665,E2 16335.665} C_VEL
LIN {X 0,Y 280.925,Z 921.601,A -85,B 0,C 180,E1 16342.865,E2 16342.865} C_VEL
LIN {X 0,Y 290.72,Z 901.782,A -85,B 0,C 180,E1 16349.702,E2 16349.702} C_VEL
LIN {X 0,Y 302.439,Z 877.167,A -85,B 0,C 180,E1 16355.465,E2 16355.465} C_VEL
LIN {X 0,Y 314.516,Z 848.603,A -85,B 0,C 180,E1 16360.067,E2 16360.067} C_VEL
LIN {X 0,Y 325.68,Z 817.07,A -85,B 0,C 180,E1 16363.604,E2 16363.604} C_VEL
LIN {X 0,Y 326.195,Z 811.534,A -85,B 0,C 180,E1 16364.427,E2 16364.427} C_VEL
LIN {X 0,Y 321.856,Z 789.372,A -85,B 0,C 180,E1 16369.215,E2 16369.215} C_VEL
LIN {X 0,Y 316.083,Z 771.647,A -85,B 0,C 180,E1 16374.137,E2 16374.137} C_VEL
LIN {X 0,Y 310.342,Z 758.697,A -85,B 0,C 180,E1 16379.413,E2 16379.413} C_VEL
LIN {X 0,Y 308.154,Z 754.098,A -85,B 0,C 180,E1 16382.017,E2 16382.017} C_VEL
LIN {X 0,Y 306.255,Z 748.94,A -85,B 0,C 180,E1 16385.677,E2 16385.677} C_VEL
LIN {X 0,Y 305.942,Z 749.568,A -85,B 0,C 180,E1 16394.662,E2 16394.662} C_VEL
